# B&R Automation Studio project mappFramework (part 11)

#### Set_AuditMgr.c
```c
#include <bur/plctypes.h>
#include <fileio.h>

#ifdef _DEFAULT_INCLUDES
#include <AsDefault.h>
#endif

#include "UnitTest.h"
#include <stdbool.h>
#include <string.h>
#include <stdlib.h>

#define TIMEOUT_TEST_CASE									\
	if (cycleCount >= 1000)									\
	{														\
		char abortMessage[80];								\
		char substate[10];									\
		memset(abortMessage, 0, sizeof(abortMessage));		\
		memset(substate, 0, sizeof(substate));				\
		itoa(TestState, substate, 10);						\
		strcpy(abortMessage, "Timeout in State = ");		\
		strcat(abortMessage, substate);						\
		TEST_FAIL(abortMessage);							\
		TEST_DONE;											\
	}

_SETUP_SET(void)
{
	cycleCount = 0;

	TEST_DONE;
}

_TEARDOWN_SET(void)
{
	TEST_DONE;
}

_SETUP_TEST(void)
{
	ArrangeDelay = 0;
	ActDelay = 0;
	AssertDelay = 0;
	ArrangeSubState = 0;
	ActSubState = 0;
	AssertSubState = 0;
	SampleTemperature = 1;
	TestComparisonNumber = 0;
	TestState = TEST_ARRANGE;
	cycleCount = 0;

	TEST_DONE;
}

_TEARDOWN_TEST(void)
{
	ArrangeDelay = 0;
	ActDelay = 0;
	AssertDelay = 0;
	SampleTemperature = 1;
	TEST_DONE;
}

_CYCLIC_SET(void)
{
	cycleCount++;
}

_TEST ExportArchive(void)
{
	TIMEOUT_TEST_CASE;

	DirInfo_0.enable = 1;
	DirInfo_0.pDevice = (UDINT) "mappAuditFiles";
	DirInfo_0.pPath = 0;
	DirInfo(&DirInfo_0);

	switch (TestState)
	{
		case TEST_ARRANGE:
			// Force an audit to be generated
			switch (ArrangeSubState)
			{
				case 0:
					SampleTemperature++;
					TEST_BUSY_CONDITION(!HmiAudit.Status.ArchiveAvailable);
					ArrangeSubState = 1;
					break;

				case 1:
					ArrangeDelay += 1;												// This delay is compensating for the function block refreshing after finishing a command
					TEST_BUSY_CONDITION(ArrangeDelay <= DelayCycles);
					TestComparisonNumber = DirInfo_0.filenum;
					TestState = TEST_ACT;
					break;
			}
			break;

		case TEST_ACT:
			// Archive audit
			switch (ActSubState)
			{
				case 0:
					HmiAudit.Commands.ExportArchives = 1;
					TEST_ABORT_CONDITION(MpAuditTrailError);
					TEST_BUSY_CONDITION(!MpAuditTrailCmdDone);
					HmiAudit.Commands.ExportArchives = 0;
					ActSubState = 1;
					break;

				case 1:
					ActDelay += 1;													// This delay is compensating for the function block refreshing after finishing a command
					TEST_BUSY_CONDITION(ActDelay <= DelayCycles);
					TestState = TEST_ASSERT;
					break;
			}
			break;

		case TEST_ASSERT:
			TEST_ASSERT(TestComparisonNumber  < DirInfo_0.filenum);
			TEST_DONE;
			break;
	}

	TEST_BUSY;
}

_TEST AutomaticArchive(void)
{
	TIMEOUT_TEST_CASE;

	switch (TestState)
	{
		case TEST_ARRANGE:
			// Set automatic archive parameters prepare audit for generation
			switch (ArrangeSubState)
			{
				case 0:
					HmiAudit.Parameters.ArchiveSettings.Enable = 1;
					HmiAudit.Parameters.ArchiveSettings.FileType = mpAUDIT_FILE_TYPE_XML;
					HmiAudit.Parameters.ArchiveSettings.MaxSize = MAX_FILE_SIZE;
					HmiAudit.Parameters.ArchiveSettings.Mode = mpAUDIT_ARCHIVE_DAILY;
					HmiAudit.Parameters.ArchiveSettings.Hour = HOUR;
					HmiAudit.Parameters.ArchiveSettings.Minute = MINUTE;
					ArrangeSubState = 1;
					break;

				case 1:
					TestComparisonNumber = HmiAudit.Status.NumberOfArchives;
					ArrangeSubState = 2;
					break;

				case 2:
					ArrangeDelay += 1;
					TEST_BUSY_CONDITION(ArrangeDelay <= DelayCycles);
					TestState = TEST_ACT;
					break;
			}
			break;

		case TEST_ACT:
			// Archive audit
			switch (ActSubState)
			{
				case 0:
					SampleTemperature = SAMPLE_TEMP_VALUE;
					DTSetTime_0.DT1 = SET_TIME;
					DTSetTime_0.enable = 1;
					DTSetTime(&DTSetTime_0);
					ActSubState = 1;
					break;

				case 1:
					TON_0.PT = TIMER_LENGTH;
					TON_0.IN = 1;
					TON(&TON_0);
					if(TON_0.Q)
					{
						ActSubState = 2;
					}
					break;

				case 2:
					TestState = TEST_ASSERT;
					TON_0.IN = 0;
					TON(&TON_0);
					break;
			}
			break;

		case TEST_ASSERT:
			// Check save location for archive
			TEST_ASSERT(TestComparisonNumber + 1 <= HmiAudit.Status.NumberOfArchives);
			TEST_DONE;
			break;
	}
	TEST_BUSY;
}

/*
B+R UnitTest: This is generated code.
Do not edit! Do not move!
Description: UnitTest Testprogramm infrastructure (TestSet).
LastUpdated: 2023-02-06 16:23:26Z
By B+R UnitTest Helper Version: 2.0.1.59
*/
UNITTEST_FIXTURES(fixtures)
{
	new_TestFixture("ExportArchive", ExportArchive),
	new_TestFixture("AutomaticArchive", AutomaticArchive),
};

UNITTEST_CALLER_COMPLETE_EXPLICIT(Set_AuditMgr, "Set_AuditMgr", setupTest, teardownTest, fixtures, setupSet, teardownSet, cyclicSetCaller);
```

- Set_Common.c (reference to Logical/UnitTestVC4/Common/CommonUT/Set_Common.c)

### Package Logical/UnitTestVC4/AppAxis_1 - Package for mapp App_Axis1 Framework

### Program Logical/UnitTestVC4/AppAxis_1/AppAxisUnitTest (ANSIC) - Unit Tests for AppAxis_1

#### variables.var
```iecst
(********************************************************************
 * COPYRIGHT --
 ********************************************************************
 * Program: utTemplate_automated
 * File: variables.var
 * Author: -
 * Created: -
 ********************************************************************
 * Local variables of program utTemplate_automated
 ********************************************************************)
(*Describe the test*)
VAR
	Testsuite : UtMgrTestSuite := (Name:='AppAxis_1VC4',Description:='AppAxis_1 VC4 Unit Tests',MetaInformation:='Meta');
END_VAR
(*Variables used in the tests*)
VAR
	MpAlarmXListUIConnect : MpAlarmXListUIConnectType := (0); (*AlarmX list connection to the UI*)
	MpAlarmXListUI_0 : MpAlarmXListUI; (*MpAlarmXList instance*)
	MpAlarmXAcknowledgeAll_0 : MpAlarmXAcknowledgeAll;
	StartingActiveAlarms : UDINT;
	StartingPendingAlarms : UDINT;
	cycleCount : USINT;
	StartPosition : LREAL;
	maxVelocity : REAL;
END_VAR
```

#### autoGeneratedFile.c
```c
/*
B+R UnitTest: This is generated code.
Do not edit! Do not move!
Description: UnitTest Testprogramm infrastructure (List of TestSets).
LastUpdated: 2022-11-08 14:30:25Z
By B+R UnitTest Helper Version: 2.0.1.59
*/
#include "UnitTest.h"

UNITTEST_TESTSET_DECLARATION  Set_Common;
UNITTEST_TESTSET_DECLARATION  Set_ManualTests;
UNITTEST_TESTSET_DECLARATION  Set_AutomaticTests;

UNITTEST_TESTSET_FIXTURES(utTestSets)
{
	new_TestSet(Set_Common),
	new_TestSet(Set_ManualTests),
	new_TestSet(Set_AutomaticTests),
};
UNTITTEST_TESTSET_HANDLER();
```

#### Set_AutomaticTests.c
```c
#include <bur/plctypes.h>

#ifdef _DEFAULT_INCLUDES
#include <AsDefault.h>
#endif

#include "UnitTest.h"
#include <stdbool.h>
#include <string.h>
#include <math.h>
#include <stdlib.h>

#define MAX(x, y) (((x) > (y)) ? (x) : (y))

#define TIMEOUT_TEST_CASE									\
	if (cycleCount >= 254)									\
	{														\
		char abortMessage[80];								\
		char substate[10];									\
		memset(abortMessage, 0, sizeof(abortMessage));		\
		memset(substate, 0, sizeof(substate));				\
		itoa(ActSubState, substate, 10);					\
		strcpy(abortMessage, "Timeout in ActSubState = ");	\
		strcat(abortMessage, substate);						\
		TEST_FAIL(abortMessage);							\
		TEST_DONE;											\
	}

_SETUP_SET(void)
{
	TEST_DONE;
}

_TEARDOWN_SET(void)
{
	TEST_DONE;
}

_SETUP_TEST(void)
{
	cycleCount = 0;
	ArrangeSubState = 0;
	ActSubState = 0;
	AssertSubState = 0;
	TestState = TEST_ARRANGE;

	maxVelocity = 0.0;
	TEST_DONE;
}

_TEARDOWN_TEST(void)
{
	AxisControl.Command.JogNegative = false;
	AxisControl.Command.JogPositive = false;
	AxisControl.Command.Abort = false;
	AxisControl.Command.LoadRecipeParameters = false;
	AxisControl.Command.MoveAbsolute = false;
	AxisControl.Command.MoveAdditive = false;
	AxisControl.Command.MoveToStart = false;
	AxisControl.Command.MoveVelocity = false;
	AxisControl.Command.Reference = false;
	AxisControl.Command.Reset = false;
	AxisControl.Command.SaveRecipeParameters = false;
	AxisControl.Command.Start = false;
	AxisControl.Command.Stop = false;
	AxisControl.Command.UpdatePreviewParameters = false;
	AxisControl.Command.UpdateVelocity = false;

	if ((AxisControl.Status.ErrorActive == true) || (MpAlarmXCoreAxis.PendingAlarms > 0))
	{
		AxisControl.Command.Reset = true;
		MpAlarmXAcknowledgeAll_0.Execute = true;
	}
	TEST_BUSY_CONDITION(AxisControl.Status.ErrorActive);
	AxisControl.Command.Reset = false;
	if (abs(AxisControl.Status.Velocity) > 0.01)
		AxisControl.Command.Stop = true;
	TEST_BUSY_CONDITION(abs(AxisControl.Status.Velocity > 0.01));
	TEST_BUSY_CONDITION(AxisControl.Status.Busy);
	AxisControl.Command.Stop = false;

	TEST_DONE;
}

_CYCLIC_SET(void)
{
	cycleCount++;
	MpAlarmXAcknowledgeAll_0.MpLink = &gMpLinkAlarmXCoreAppAxis_1;
	MpAlarmXAcknowledgeAll_0.Enable = true;
	MpAlarmXAcknowledgeAll(&MpAlarmXAcknowledgeAll_0);
	MpAlarmXAcknowledgeAll_0.Execute = false;
}

_TEST Start(void)
{
	TIMEOUT_TEST_CASE
	switch (TestState)
	{
		case TEST_ARRANGE:
			AxisControl.Parameters.Velocity = 40;
			TestState = TEST_ACT;
			break;

		case TEST_ACT:
			maxVelocity = MAX(AxisControl.Status.Velocity, maxVelocity);
			switch (ActSubState)
			{
				case 0:
					AxisControl.Command.Start = true;
					TEST_BUSY_CONDITION(!AxisControl.Status.Busy);
					ActSubState = 1;
					break;

				case 1:
					TEST_BUSY_CONDITION(cycleCount < 30);
					TestState = TEST_ASSERT;
					break;
			}
			break;

		case TEST_ASSERT:
			TEST_ASSERT_FLOAT_WITHIN(0.1, 40.0, maxVelocity);
			TEST_DONE;
			break;
	}
	TEST_BUSY;
}

_TEST UpdateVelocity(void)
{
	TIMEOUT_TEST_CASE
	switch (TestState)
	{
		case TEST_ARRANGE:
			AxisControl.Parameters.Velocity = 40;
			TestState = TEST_ACT;
			break;

		case TEST_ACT:
			maxVelocity = MAX(AxisControl.Status.Velocity, maxVelocity);
			switch (ActSubState)
			{
				case 0:
					AxisControl.Command.Start = true;
					TEST_BUSY_CONDITION(!AxisControl.Status.Busy);
					ActSubState = 1;
					break;

				case 1:
					TEST_BUSY_CONDITION(cycleCount < 30);
					TEST_ASSERT_FLOAT_WITHIN(0.1, 40.0, maxVelocity);
					AxisControl.Command.UpdateVelocity = true;
					AxisControl.Parameters.Velocity = 60;
					ActSubState = 2;
					break;

				case 2:
					TEST_BUSY_CONDITION(cycleCount < 60);
					TestState = TEST_ASSERT;
					break;
			}
			break;

		case TEST_ASSERT:
			TEST_ASSERT_FLOAT_WITHIN(0.1, 60.0, maxVelocity);
			TEST_DONE;
			break;
	}
	TEST_BUSY;
}

_TEST ZeroVelocity(void)
{
	TIMEOUT_TEST_CASE
	switch (TestState)
	{
		case TEST_ARRANGE:
			AxisControl.Parameters.Velocity = 0;
			TestState = TEST_ACT;
			break;

		case TEST_ACT:
			maxVelocity = MAX(AxisControl.Status.Velocity, maxVelocity);
			switch (ActSubState)
			{
				case 0:
					AxisControl.Command.Start = true;
					TEST_BUSY_CONDITION(!AxisControl.Status.Busy);
					ActSubState = 1;
					break;

				case 1:
					TEST_BUSY_CONDITION(cycleCount < 10);
					TestState = TEST_ASSERT;
					break;
			}
			break;

		case TEST_ASSERT:
			TEST_ASSERT(AxisControl.Status.ErrorActive);
			TEST_ASSERT_EQUAL_INT(1, MpAlarmXCoreAxis.PendingAlarms);
			TEST_ASSERT_FLOAT_WITHIN(0.1, 0.0, maxVelocity);
			TEST_DONE;
			break;
	}
	TEST_BUSY;
}

/*
B+R UnitTest: This is generated code.
Do not edit! Do not move!
Description: UnitTest Testprogramm infrastructure (TestSet).
LastUpdated: 2022-11-08 14:33:54Z
By B+R UnitTest Helper Version: 2.0.1.59
*/
UNITTEST_FIXTURES(fixtures)
{
	new_TestFixture("Start", Start),
	new_TestFixture("UpdateVelocity", UpdateVelocity),
	new_TestFixture("ZeroVelocity", ZeroVelocity),
};

UNITTEST_CALLER_COMPLETE_EXPLICIT(Set_AutomaticTests, "Set_AutomaticTests", setupTest, teardownTest, fixtures, setupSet, teardownSet, cyclicSetCaller);
```

#### Set_ManualTests.c
```c
#include <bur/plctypes.h>

#ifdef _DEFAULT_INCLUDES
#include <AsDefault.h>
#endif

#include "UnitTest.h"
#include <stdbool.h>
#include <string.h>
#include <math.h>
#include <stdlib.h>

#define MAX(x, y) (((x) > (y)) ? (x) : (y))

#define TIMEOUT_TEST_CASE									\
	if (cycleCount >= 254)									\
	{														\
		char abortMessage[80];								\
		char substate[10];									\
		memset(abortMessage, 0, sizeof(abortMessage));		\
		memset(substate, 0, sizeof(substate));				\
		itoa(ActSubState, substate, 10);					\
		strcpy(abortMessage, "Timeout in ActSubState = ");	\
		strcat(abortMessage, substate);						\
		TEST_FAIL(abortMessage);							\
		TEST_DONE;											\
	}

_SETUP_SET(void)
{
	TEST_DONE;
}

_TEARDOWN_SET(void)
{
	TEST_DONE;
}

_SETUP_TEST(void)
{
	cycleCount = 0;
	ArrangeSubState = 0;
	ActSubState = 0;
	AssertSubState = 0;
	TestState = TEST_ARRANGE;

	maxVelocity = 0.0;

	TEST_DONE;
}

_TEARDOWN_TEST(void)
{
	AxisControl.Command.JogNegative = false;
	AxisControl.Command.JogPositive = false;
	AxisControl.Command.Abort = false;
	AxisControl.Command.LoadRecipeParameters = false;
	AxisControl.Command.MoveAbsolute = false;
	AxisControl.Command.MoveAdditive = false;
	AxisControl.Command.MoveToStart = false;
	AxisControl.Command.MoveVelocity = false;
	AxisControl.Command.Reference = false;
	AxisControl.Command.Reset = false;
	AxisControl.Command.SaveRecipeParameters = false;
	AxisControl.Command.Start = false;
	AxisControl.Command.Stop = false;
	AxisControl.Command.UpdatePreviewParameters = false;
	AxisControl.Command.UpdateVelocity = false;

	if ((AxisControl.Status.ErrorActive == true) || (MpAlarmXCoreAxis.PendingAlarms > 0))
	{
		AxisControl.Command.Reset = true;
		MpAlarmXAcknowledgeAll_0.Execute = true;
	}
	TEST_BUSY_CONDITION(AxisControl.Status.ErrorActive);
	AxisControl.Command.Reset = false;
	if (abs(AxisControl.Status.Velocity) > 0.01)
		AxisControl.Command.Stop = true;
	TEST_BUSY_CONDITION(abs(AxisControl.Status.Velocity > 0.01));
	TEST_BUSY_CONDITION(AxisControl.Status.Busy);
	AxisControl.Command.Stop = false;

	TEST_DONE;
}

_CYCLIC_SET(void)
{
	cycleCount++;

	MpAlarmXListUI_0.Enable = true;
	MpAlarmXListUI_0.UIConnect = &MpAlarmXListUIConnect;
	MpAlarmXListUI_0.MpLink = &gMpLinkAlarmXCoreAppAxis_1;
	MpAlarmXListUI_0.UISetup.AlarmListScrollWindow = 10;
	MpAlarmXListUI_0.UISetup.AlarmListSize = 50;
	strcpy(MpAlarmXListUI_0.UISetup.TimeStampPattern, "%Y %m %d %H:%M:%S");
	MpAlarmXListUI(&MpAlarmXListUI_0);

	MpAlarmXAcknowledgeAll_0.MpLink = &gMpLinkAlarmXCoreAppAxis_1;
	MpAlarmXAcknowledgeAll_0.Enable = true;
	MpAlarmXAcknowledgeAll(&MpAlarmXAcknowledgeAll_0);
	TEST_BUSY_CONDITION(MpAlarmXAcknowledgeAll_0.CommandBusy);
	MpAlarmXAcknowledgeAll_0.Execute = false;

}

_TEST PowerOn(void)
{
	TIMEOUT_TEST_CASE
	switch (TestState)
	{
		case TEST_ARRANGE:
			TestState = TEST_ACT;
			break;

		case TEST_ACT:
			switch (ActSubState)
			{
				case 0:
					AxisControl.Command.Power = true;
					ActSubState = 1;
					break;
				case 1:
					TEST_BUSY_CONDITION(AxisControl.Status.Busy == true);
					TestState = TEST_ASSERT;
					break;
			}
			break;

		case TEST_ASSERT:
			TEST_ASSERT(AxisControl.Status.IsPowered);
			TEST_DONE;
			break;
	}
	TEST_BUSY;
}

_TEST Homing(void)
{
	TIMEOUT_TEST_CASE
	switch (TestState)
	{
		case TEST_ARRANGE:
			TestState = TEST_ACT;
			break;

		case TEST_ACT:
			switch (ActSubState)
			{
				case 0:
					AxisControl.Command.Reference = true;
					ActSubState = 1;
					break;
				case 1:
					TEST_BUSY_CONDITION(AxisControl.Status.IsHomed == false);
					TEST_BUSY_CONDITION(!AxisControl.Status.Busy);
					ActSubState = 2;
					break;

				case 2:
					TEST_BUSY_CONDITION(AxisControl.Status.Busy);
					TestState = TEST_ASSERT;
					break;
			}
			break;

		case TEST_ASSERT:
			TEST_ASSERT(AxisControl.Status.IsHomed);
			TEST_ASSERT_DOUBLE_WITHIN(0.0001, 0.0, AxisControl.Status.Position);
			TEST_DONE;
			break;
	}
	TEST_BUSY;
}

_TEST JogPositive(void)
{
	TIMEOUT_TEST_CASE
	switch (TestState)
	{
		case TEST_ARRANGE:
			TestState = TEST_ACT;
			break;

		case TEST_ACT:
			switch (ActSubState)
			{
				case 0:
					AxisControl.Command.JogPositive = true;
					AxisControl.Parameters.JogVelocity = 50;
					ActSubState = 1;
					break;
				case 1:
					TEST_BUSY_CONDITION(AxisControl.Status.Velocity <= 49.0);
					TestState = TEST_ASSERT;
					break;
			}
			break;

		case TEST_ASSERT:
			TEST_ASSERT_FLOAT_WITHIN(0.1, 50.0, AxisControl.Status.Velocity);
			TEST_DONE;
			break;
	}
	TEST_BUSY;
}

_TEST JogNegative(void)
{
	TIMEOUT_TEST_CASE
	switch (TestState)
	{
		case TEST_ARRANGE:
			TestState = TEST_ACT;
			break;

		case TEST_ACT:
			switch (ActSubState)
			{
				case 0:
					AxisControl.Command.JogNegative = true;
					AxisControl.Parameters.JogVelocity = 50;
					ActSubState = 1;
					break;
				case 1:
					TEST_BUSY_CONDITION(AxisControl.Status.Velocity >= -49.0);
					TestState = TEST_ASSERT;
					break;
			}
			break;

		case TEST_ASSERT:
			TEST_ASSERT_FLOAT_WITHIN(0.1, -50.0, AxisControl.Status.Velocity);
			TEST_DONE;
			break;
	}
	TEST_BUSY;
}

_TEST MoveAbsolute(void)
{
	TIMEOUT_TEST_CASE
	switch (TestState)
	{
		case TEST_ARRANGE:
			AxisControl.Parameters.Position = 10;
			AxisControl.Parameters.Velocity = 40;
			TestState = TEST_ACT;
			break;

		case TEST_ACT:
			maxVelocity = MAX(AxisControl.Status.Velocity, maxVelocity);
			switch (ActSubState)
			{
				case 0:
					AxisControl.Command.MoveAbsolute = true;
					TEST_BUSY_CONDITION(!AxisControl.Status.Busy);
					ActSubState = 1;
					break;
				case 1:
					TEST_BUSY_CONDITION(AxisControl.Status.Busy);
					AxisControl.Command.MoveAbsolute = false;
					TestState = TEST_ASSERT;
					break;
			}
			break;

		case TEST_ASSERT:
			TEST_ASSERT_FLOAT_WITHIN(0.1, 40.0, maxVelocity);
			TEST_ASSERT_FLOAT_WITHIN(0.01, 10.0, AxisControl.Status.Position);
			TEST_DONE;
			break;
	}
	TEST_BUSY;
}

_TEST MoveAdditive(void)
{
	TIMEOUT_TEST_CASE
	switch (TestState)
	{
		case TEST_ARRANGE:
			AxisControl.Parameters.Distance = 5;
			AxisControl.Parameters.Velocity = 30;
			StartPosition = AxisControl.Status.Position;
			TestState = TEST_ACT;
			break;

		case TEST_ACT:
			maxVelocity = MAX(AxisControl.Status.Velocity, maxVelocity);
			switch (ActSubState)
			{
				case 0:
					AxisControl.Command.MoveAdditive = true;
					TEST_BUSY_CONDITION(!AxisControl.Status.Busy);
					ActSubState = 1;
					break;
				case 1:
					TEST_BUSY_CONDITION(AxisControl.Status.Busy);
					AxisControl.Command.MoveAbsolute = false;
					TestState = TEST_ASSERT;
					break;
			}
			break;

		case TEST_ASSERT:
			TEST_ASSERT_FLOAT_WITHIN(0.1, 30.0, maxVelocity);
			TEST_ASSERT_FLOAT_WITHIN(0.01, StartPosition + 5.0, AxisControl.Status.Position);
			TEST_DONE;
			break;
	}
	TEST_BUSY;
}

_TEST MoveVelocity(void)
{
	TIMEOUT_TEST_CASE
	switch (TestState)
	{
		case TEST_ARRANGE:
			AxisControl.Parameters.Velocity = 25;
			TestState = TEST_ACT;
			break;

		case TEST_ACT:
			maxVelocity = MAX(AxisControl.Status.Velocity, maxVelocity);
			switch (ActSubState)
			{
				case 0:
					AxisControl.Command.MoveVelocity = true;
					TEST_BUSY_CONDITION(!AxisControl.Status.Busy);
					ActSubState = 1;
					break;
				case 1:
					TEST_BUSY_CONDITION(cycleCount < 30);
					TestState = TEST_ASSERT;
					break;
			}
			break;

		case TEST_ASSERT:
			TEST_ASSERT_FLOAT_WITHIN(0.1, 25.0, maxVelocity);
			TEST_DONE;
			break;
	}
	TEST_BUSY;
}

_TEST MoveJogPositiveStop(void)
{
	TIMEOUT_TEST_CASE
	switch (TestState)
	{
		case TEST_ARRANGE:
			AxisControl.Parameters.JogVelocity = 25;
			TestState = TEST_ACT;
			break;

		case TEST_ACT:
			maxVelocity = MAX(AxisControl.Status.Velocity, maxVelocity);
			switch (ActSubState)
			{
				case 0:
					AxisControl.Command.JogPositive = true;
					TEST_BUSY_CONDITION(!AxisControl.Status.Busy);
					ActSubState = 1;
					break;
				case 1:
					TEST_BUSY_CONDITION(cycleCount < 30);
					AxisControl.Command.JogPositive = false;
					ActSubState = 2;
					break;
				case 2:
					TEST_BUSY_CONDITION(AxisControl.Status.Busy);
					TestState = TEST_ASSERT;
					break;
			}
			break;

		case TEST_ASSERT:
			TEST_ASSERT_FLOAT_WITHIN(0.1, 0.0, AxisControl.Status.Velocity);
			TEST_DONE;
			break;
	}
	TEST_BUSY;
}

_TEST MoveJogNegativeStop(void)
{
	TIMEOUT_TEST_CASE
	switch (TestState)
	{
		case TEST_ARRANGE:
			AxisControl.Parameters.JogVelocity = 25;
			TestState = TEST_ACT;
			break;

		case TEST_ACT:
			maxVelocity = MAX(AxisControl.Status.Velocity, maxVelocity);
			switch (ActSubState)
			{
				case 0:
					AxisControl.Command.JogNegative = true;
					TEST_BUSY_CONDITION(!AxisControl.Status.Busy);
					ActSubState = 1;
					break;
				case 1:
					TEST_BUSY_CONDITION(cycleCount < 30);
					AxisControl.Command.JogNegative = false;
					ActSubState = 2;
					break;
				case 2:
					TEST_BUSY_CONDITION(AxisControl.Status.Busy);
					TestState = TEST_ASSERT;
					break;
			}
			break;

		case TEST_ASSERT:
			TEST_ASSERT_FLOAT_WITHIN(0.1, 0.0, AxisControl.Status.Velocity);
			TEST_DONE;
			break;
	}
	TEST_BUSY;
}

_TEST MoveAbsoluteStop(void)
{
	TIMEOUT_TEST_CASE
	switch (TestState)
	{
		case TEST_ARRANGE:
			AxisControl.Parameters.Position = 1;
			AxisControl.Parameters.Velocity = 25;
			TestState = TEST_ACT;
			break;

		case TEST_ACT:
			maxVelocity = MAX(AxisControl.Status.Velocity, maxVelocity);
			switch (ActSubState)
			{
				case 0:
					AxisControl.Command.MoveAbsolute = true;
					TEST_BUSY_CONDITION(!AxisControl.Status.Busy);
					ActSubState = 1;
					break;
				case 1:
					TEST_BUSY_CONDITION(cycleCount < 30);
					AxisControl.Command.MoveAbsolute = false;
					AxisControl.Command.Stop = true;
					ActSubState = 2;
					break;
				case 2:
					TEST_BUSY_CONDITION(AxisControl.Status.Busy);
					TestState = TEST_ASSERT;
					break;
			}
			break;

		case TEST_ASSERT:
			TEST_ASSERT_FLOAT_WITHIN(0.1, 0.0, AxisControl.Status.Velocity);
			// check that we are not at the target position
			TEST_ASSERT(fabs(1.0 - AxisControl.Status.Position) > 0.01);
			TEST_DONE;
			break;
	}
	TEST_BUSY;
}

_TEST MoveAdditiveStop(void)
{
	TIMEOUT_TEST_CASE
	switch (TestState)
	{
		case TEST_ARRANGE:
			AxisControl.Parameters.Distance = 10;
			AxisControl.Parameters.Velocity = 25;
			StartPosition = AxisControl.Status.Position;
			TestState = TEST_ACT;
			break;

		case TEST_ACT:
			maxVelocity = MAX(AxisControl.Status.Velocity, maxVelocity);
			switch (ActSubState)
			{
				case 0:
					AxisControl.Command.MoveAdditive = true;
					TEST_BUSY_CONDITION(!AxisControl.Status.Busy);
					ActSubState = 1;
					break;
				case 1:
					TEST_BUSY_CONDITION(cycleCount < 30);
					AxisControl.Command.MoveAdditive = false;
					AxisControl.Command.Stop = true;
					ActSubState = 2;
					break;
				case 2:
					TEST_BUSY_CONDITION(AxisControl.Status.Busy);
					TestState = TEST_ASSERT;
					break;
			}
			break;

		case TEST_ASSERT:
			TEST_ASSERT_FLOAT_WITHIN(0.1, 0.0, AxisControl.Status.Velocity);
			// check that we are not at the target position
			TEST_ASSERT(fabs((StartPosition + 10.0) - AxisControl.Status.Position) > 0.01);
			TEST_DONE;
			break;
	}
	TEST_BUSY;
}

_TEST MoveVelocityStop(void)
{
	TIMEOUT_TEST_CASE
	switch (TestState)
	{
		case TEST_ARRANGE:
			AxisControl.Parameters.Velocity = 25;
			TestState = TEST_ACT;
			break;

		case TEST_ACT:
			maxVelocity = MAX(AxisControl.Status.Velocity, maxVelocity);
			switch (ActSubState)
			{
				case 0:
					AxisControl.Command.MoveVelocity = true;
					TEST_BUSY_CONDITION(!AxisControl.Status.Busy);
					ActSubState = 1;
					break;
				case 1:
					TEST_BUSY_CONDITION(cycleCount < 30);
					AxisControl.Command.MoveVelocity = false;
					AxisControl.Command.Stop = true;
					ActSubState = 2;
					break;
				case 2:
					TEST_BUSY_CONDITION(AxisControl.Status.Busy);
					TestState = TEST_ASSERT;
					break;
			}
			break;

		case TEST_ASSERT:
			TEST_ASSERT_FLOAT_WITHIN(0.1, 0.0, AxisControl.Status.Velocity);
			TEST_DONE;
			break;
	}
	TEST_BUSY;
}

_TEST TriggerAlarm(void)
{
	TIMEOUT_TEST_CASE
	switch (TestState)
	{
		case TEST_ARRANGE:
			AxisControl.Parameters.Velocity = 10001;
			TestState = TEST_ACT;
			break;

		case TEST_ACT:
			maxVelocity = MAX(AxisControl.Status.Velocity, maxVelocity);
			switch (ActSubState)
			{
				case 0:
					AxisControl.Command.MoveVelocity = true;
					TEST_BUSY_CONDITION(!AxisControl.Status.Busy);
					ActSubState = 1;
					break;
				case 1:
					TEST_BUSY_CONDITION(cycleCount < 20);
					TestState = TEST_ASSERT;
					break;
			}
			break;

		case TEST_ASSERT:
			TEST_ASSERT_FLOAT_WITHIN(0.1, 0.0, AxisControl.Status.Velocity);
			TEST_ASSERT_FLOAT_WITHIN(0.1, 0.0, maxVelocity);
			TEST_ASSERT(AxisControl.Status.ErrorActive);
			TEST_ASSERT_EQUAL_INT(1, MpAlarmXCoreAxis.PendingAlarms);
			TEST_DONE;
			break;
	}
	TEST_BUSY;
}

_TEST ResetAlarm(void)
{
	TIMEOUT_TEST_CASE
	switch (TestState)
	{
		case TEST_ARRANGE:
			AxisControl.Parameters.Velocity = 10001;
			StartingPendingAlarms = MpAlarmXCoreAxis.PendingAlarms;
			TestState = TEST_ACT;
			break;

		case TEST_ACT:
			maxVelocity = MAX(AxisControl.Status.Velocity, maxVelocity);
			switch (ActSubState)
			{
				case 0:
					AxisControl.Command.MoveVelocity = true;
					TEST_BUSY_CONDITION(!AxisControl.Status.Busy);
					ActSubState = 1;
					break;
				case 1:
					TEST_BUSY_CONDITION(!AxisControl.Status.ErrorActive);
					TEST_BUSY_CONDITION(MpAlarmXCoreAxis.PendingAlarms == StartingPendingAlarms);
					AxisControl.Command.MoveVelocity = false;
					ActSubState = 2;
					break;
				case 2:
					// wait until the command is received by the axis task
					TEST_BUSY_CONDITION(State != STATE_RESETTING);
					AxisControl.Command.Reset = true;
					MpAlarmXAcknowledgeAll_0.Execute = true;
					ActSubState = 3;
					break;
				case 3:
					TEST_BUSY_CONDITION(AxisControl.Status.Busy);
					TestState = TEST_ASSERT;
					break;
			}
			break;

		case TEST_ASSERT:
			TEST_ASSERT(!AxisControl.Status.ErrorActive);
			TEST_ASSERT_EQUAL_INT(0, MpAlarmXCoreAxis.PendingAlarms);
			TEST_DONE;
			break;
	}
	TEST_BUSY;
}

_TEST UpdateVelocity(void)
{
	TIMEOUT_TEST_CASE
	switch (TestState)
	{
		case TEST_ARRANGE:
			AxisControl.Parameters.Velocity = 40;
			TestState = TEST_ACT;
			break;

		case TEST_ACT:
			maxVelocity = MAX(AxisControl.Status.Velocity, maxVelocity);
			switch (ActSubState)
			{
				case 0:
					AxisControl.Command.MoveVelocity = true;
					TEST_BUSY_CONDITION(!AxisControl.Status.Busy);
					ActSubState = 1;
					break;
				case 1:
					TEST_BUSY_CONDITION(cycleCount < 30);
					TEST_ASSERT_FLOAT_WITHIN(0.1, 40.0, maxVelocity);
					AxisControl.Command.UpdateVelocity = true;
					AxisControl.Parameters.Velocity = 60;
					ActSubState = 2;
					break;
				case 2:
					TEST_BUSY_CONDITION(cycleCount < 60);
					TestState = TEST_ASSERT;
					break;
			}
			break;

		case TEST_ASSERT:
			// update velocity should not affect manual moves
			TEST_ASSERT_FLOAT_WITHIN(0.1, 40.0, maxVelocity);
			TEST_DONE;
			break;
	}
	TEST_BUSY;
}

/*
B+R UnitTest: This is generated code.
Do not edit! Do not move!
Description: UnitTest Testprogramm infrastructure (TestSet).
LastUpdated: 2022-11-15 16:02:39Z
By B+R UnitTest Helper Version: 2.0.1.59
*/
UNITTEST_FIXTURES(fixtures)
{
	new_TestFixture("PowerOn", PowerOn),
	new_TestFixture("Homing", Homing),
	new_TestFixture("JogPositive", JogPositive),
	new_TestFixture("JogNegative", JogNegative),
	new_TestFixture("MoveAbsolute", MoveAbsolute),
	new_TestFixture("MoveAdditive", MoveAdditive),
	new_TestFixture("MoveVelocity", MoveVelocity),
	new_TestFixture("MoveJogPositiveStop", MoveJogPositiveStop),
	new_TestFixture("MoveJogNegativeStop", MoveJogNegativeStop),
	new_TestFixture("MoveAbsoluteStop", MoveAbsoluteStop),
	new_TestFixture("MoveAdditiveStop", MoveAdditiveStop),
	new_TestFixture("MoveVelocityStop", MoveVelocityStop),
	new_TestFixture("TriggerAlarm", TriggerAlarm),
	new_TestFixture("ResetAlarm", ResetAlarm),
	new_TestFixture("UpdateVelocity", UpdateVelocity),
};

UNITTEST_CALLER_COMPLETE_EXPLICIT(Set_ManualTests, "Set_ManualTests", setupTest, teardownTest, fixtures, setupSet, teardownSet, cyclicSetCaller);
```

#### testSuite.c
```c
/********************************************************************
 * COPYRIGHT --
 ********************************************************************
 * Program: -
 * Author:
 * Created:
 ********************************************************************
 * Test registration and handshake
 ********************************************************************/

#include <bur/plctypes.h>

#ifdef _DEFAULT_INCLUDES
#include <AsDefault.h>
#endif

#include "UnitTest.h"
#include <string.h>
#include <stdbool.h>

void _INIT initTestSuite(void)
{
	Testsuite.Enable = 1;
	utInit(&Testsuite);

	CommonTestsuite.Enable = 1;
	utInit(&CommonTestsuite);

	strcpy((char*)&FileDeviceName, "");
	strcpy((char*)&TextNameSpace, "Axis/Alarms");
	strcpy((char*)&TextID, "ReferenceRequired");
}

void _CYCLIC cyclicWithTest(void)
{
	utCyclic(&Testsuite);

	if (Testsuite.Informational.LastKnownPassedLocation.TestCaseName != 0)
		strcpy((char*)&LastTestCase, (char*)Testsuite.Informational.LastKnownPassedLocation.TestCaseName);
	if (Testsuite.Informational.LastKnownPassedLocation.TestSetName != 0)
		strcpy((char*)&LastTestSet, (char*)Testsuite.Informational.LastKnownPassedLocation.TestSetName);
	if (Testsuite.Informational.LastKnownPassedLocation.File != 0)
		strcpy((char*)&LastTestFile, (char*)Testsuite.Informational.LastKnownPassedLocation.File);
}

void _EXIT exitTestSuite(void)
{
	utExit(&Testsuite);
}
```

### Package Logical/UnitTestVC4/Backup - Package for mapp Backup Framework

### Program Logical/UnitTestVC4/Backup/BackupUnitTest (ANSIC)

- BackupMgr.typ (reference to Logical/Infrastructure/VC4/Backup/BackupMgr/BackupMgr.typ)

- BackupMgr.var (reference to Logical/Infrastructure/VC4/Backup/BackupMgr/BackupMgr.var)

#### variables.var - Name the suite and add PVs for the program
```iecst
(********************************************************************
 * COPYRIGHT --
 ********************************************************************
 * Program: utTemplate_automated
 * File: variables.var
 * Author: -
 * Created: -
 ********************************************************************
 * Local variables of program utTemplate_automated
 ********************************************************************)
(*Describe the test*)
VAR
	Testsuite : UtMgrTestSuite := (Name:='BackupMgrVC4',Description:='BackupMgr VC4 Unit Tests',MetaInformation:='Meta');
END_VAR
(*Variables used in the tests*)
```

#### testSuite.c
```c
/********************************************************************
 * COPYRIGHT --
 ********************************************************************
 * Program: -
 * Author:
 * Created:
 ********************************************************************
 * Test registration and handshake
 ********************************************************************/

#include <bur/plctypes.h>

#ifdef _DEFAULT_INCLUDES
#include <AsDefault.h>
#endif

#include "UnitTest.h"
#include <string.h>

void _INIT initTestSuite(void)
{
	Testsuite.Enable = 1;
	utInit(&Testsuite);

	CommonTestsuite.Enable = 1;
	utInit(&CommonTestsuite);

	strcpy((char*)&FileDeviceName, "mappBackupFiles");
	strcpy((char*)&TextNameSpace, "mappFramework/Backup/Alarms");
	strcpy((char*)&TextID, "CreateFailed");

}

void _CYCLIC cyclicWithTest(void)
{
	utCyclic(&Testsuite);
}

void _EXIT exitTestSuite(void)
{
	utExit(&Testsuite);
}
```

#### Set_BackupMgr.c
```c
#include <bur/plctypes.h>

#ifdef _DEFAULT_INCLUDES
#include <AsDefault.h>
#endif

#include "UnitTest.h"
#include <stdbool.h>
#include <string.h>

_SETUP_SET(void)
{
	TEST_DONE;
}

_TEARDOWN_SET(void)
{
	TEST_DONE;
}

_SETUP_TEST(void)
{
	TEST_DONE;
}

_TEARDOWN_TEST(void)
{
	TEST_DONE;
}

/*
B+R UnitTest: This is generated code.
Do not edit! Do not move!
Description: UnitTest Testprogramm infrastructure (TestSet).
LastUpdated: 2022-09-22 14:29:52Z
By B+R UnitTest Helper Version: 2.0.1.59
*/
UNITTEST_FIXTURES(fixtures)
{
};

UNITTEST_CALLER_COMPLETE_EXPLICIT(Set_BackupMgr, "Set_BackupMgr", setupTest, teardownTest, fixtures, setupSet, teardownSet, 0);
```

- Set_Common.c (reference to Logical/UnitTestVC4/Common/CommonUT/Set_Common.c)

### Package Logical/UnitTestVC4/File - Package for mapp File Framework

### Program Logical/UnitTestVC4/File/FileUnitTest (ANSIC) - Unit Tests for FileMgr

- FileMgr.typ (reference to Logical/Infrastructure/VC4/File/FileMgr/FileMgr.typ)

- FileMgr.var (reference to Logical/Infrastructure/VC4/File/FileMgr/FileMgr.var)

- Set_Common.c (reference to Logical/UnitTestVC4/Common/CommonUT/Set_Common.c)

#### variables.var - Name the suite and add PVs for the program
```iecst
(********************************************************************
 * COPYRIGHT --
 ********************************************************************
 * Program: utTemplate_automated
 * File: variables.var
 * Author: -
 * Created: -
 ********************************************************************
 * Local variables of program utTemplate_automated
 ********************************************************************)
(*Describe the test*)
VAR
	Testsuite : UtMgrTestSuite := (Name:='FileMgrVC4',Description:='FileMgr VC4 Unit Tests',Type:=utMgrTEST_TYPE_C,MetaInformation:='Meta');
END_VAR
(*Variables used in the tests*)
VAR
	cycleCount : {REDUND_UNREPLICABLE} UINT;
	HmiFile_UT : FileHmiInterfaceType; (*HMI interface structure*)
	FileName : STRING[24];
	FileNumber : USINT;
	SetupState : USINT;
	FileCreate_UT : FileCreate;
	FileClose_UT : FileClose;
	NumberOfFiles : UINT;
	CurrentFile : UINT;
	DirInfo_UT : DirInfo;
	fileInfo : fiDIR_READ_DATA;
	DirRead_UT : DirRead;
	FileWrite_UT : FileWrite;
	testData : {REDUND_UNREPLICABLE} STRING[1023] := 'testing data';
	FileDelete_UT : FileDelete;
	NameMatch : BOOL;
	DirName : STRING[255] := 'FileTestDir';
	CreateFileName : STRING[255] := 'FileTestFile.xml';
	FileCreate_0 : FileCreate;
	FileClose_0 : FileClose;
	CopiedFileName : STRING[255] := 'FileTestFile(1).xml';
	CopiedDirName : STRING[255] := 'FileTestDir(1)';
	NewFileName : STRING[255] := 'FileRename.xml';
	NewDirName : STRING[255] := 'DirRename';
	InNewLocation : BOOL;
	InOldLocation : BOOL;
	CopiedNewFileName : STRING[255] := 'FileRename(1).xml';
	CopiedNewDirName : STRING[255] := 'DirRename(1)';
	MultiSelectFileCopy : BOOL;
	MultiSelectDirCopy : BOOL;
END_VAR
```

#### testSuite.c
```c
/********************************************************************
 * COPYRIGHT --
 ********************************************************************
 * Program: -
 * Author:
 * Created:
 ********************************************************************
 * Test registration and handshake
 ********************************************************************/

#include <bur/plctypes.h>

#ifdef _DEFAULT_INCLUDES
#include <AsDefault.h>
#endif
#include <string.h>

#include "UnitTest.h"

void _INIT initTestSuite(void)
{
	Testsuite.Enable = 1;
	utInit(&Testsuite);

	CommonTestsuite.Enable = 1;
	utInit(&CommonTestsuite);

	strcpy((char*)&TextNameSpace, "mappFramework/File/Alarms");
	strcpy((char*)&TextID, "DeviceNotFound");
	strcpy(FileDeviceName, "mappUserXFiles");
}

void _CYCLIC cyclicWithTest(void)
{
	utCyclic(&Testsuite);
	if (Testsuite.Informational.LastKnownPassedLocation.TestCaseName != 0)
		strcpy((char*)&LastTestCase, (char*)Testsuite.Informational.LastKnownPassedLocation.TestCaseName);
	if (Testsuite.Informational.LastKnownPassedLocation.TestSetName != 0)
		strcpy((char*)&LastTestSet, (char*)Testsuite.Informational.LastKnownPassedLocation.TestSetName);
	if (Testsuite.Informational.LastKnownPassedLocation.File != 0)
		strcpy((char*)&LastTestFile, (char*)Testsuite.Informational.LastKnownPassedLocation.File);
}

void _EXIT exitTestSuite(void)
{
	utExit(&Testsuite);
}
```

#### Set_FileMgr.c
```c
#include <bur/plctypes.h>

#ifdef _DEFAULT_INCLUDES
#include <AsDefault.h>
#endif

#include "UnitTest.h"
#include <stdbool.h>
#include <string.h>
#include <stdlib.h>

#define TIMEOUT_TEST_CASE								\
	if (cycleCount >= 1000)								\
	{													\
	char abortMessage[80];								\
	char substate[10];									\
	memset(abortMessage, 0, sizeof(abortMessage));		\
	memset(substate, 0, sizeof(substate));				\
	itoa(TestState, substate, 10);						\
	strcpy(abortMessage, "Timeout in State = ");		\
	strcat(abortMessage, substate);						\
	TEST_FAIL(abortMessage);							\
	TEST_DONE;											\
	}

_SETUP_SET(void)
{
	TestState = 0;
	FileNumber = 0;

	HmiFile_UT.Parameters.Fifo.Enable = false;
	HmiFile_UT.Parameters.Fifo.ScanInterval = 60;
	strcpy(HmiFile_UT.Parameters.Fifo.DeviceName, "mappUserXFiles");

	switch (SetupState)
	{
		case 0:
			TEST_BUSY_CONDITION(HmiFile_UT.Status.DeleteStep != FILE_DISABLED);
			for (USINT i=0; i<sizeof(HmiFile_UT.Status.FifoSelect)/sizeof(HmiFile_UT.Status.FifoSelect[0]); i++)
			{
				TEST_BUSY_CONDITION(HmiFile_UT.Status.FifoSelect[i] != 0);
			}

			DirInfo_UT.enable = true;
			DirInfo_UT.pDevice = (UDINT)&"mappUserXFiles";
			DirInfo_UT.pPath = (UDINT)&"";
			DirInfo(&DirInfo_UT);
			TEST_BUSY_CONDITION(DirInfo_UT.status == 65535);
			TEST_ABORT_CONDITION(DirInfo_UT.status != 0);
			NumberOfFiles = DirInfo_UT.filenum;
			CurrentFile = 0;
			SetupState = (NumberOfFiles == 0) ? 100 : 1;
			break;

		case 1:
			DirRead_UT.enable = true;
			DirRead_UT.pDevice = DirInfo_UT.pDevice;
			DirRead_UT.entry = 0;
			DirRead_UT.option = fiFILE;
			DirRead_UT.pData = (UDINT)&fileInfo;
			DirRead_UT.data_len = sizeof(fileInfo);
			DirRead(&DirRead_UT);
			TEST_BUSY_CONDITION(DirRead_UT.status == 65535);
			TEST_ABORT_CONDITION(DirRead_UT.status != 0);
			SetupState = 2;
			break;

		case 2:
			FileDelete_UT.enable = true;
			FileDelete_UT.pDevice = DirInfo_UT.pDevice;
			FileDelete_UT.pName = (UDINT)&fileInfo.Filename;
			FileDelete(&FileDelete_UT);
			TEST_BUSY_CONDITION(FileDelete_UT.status == 65535);
			TEST_ABORT_CONDITION(FileDelete_UT.status != 0);

			CurrentFile++;
			SetupState = (CurrentFile >= NumberOfFiles) ? 100 : 1;
			break;

		case 10:
			TEST_BUSY_CONDITION(MpFileManagerUIConnect_FIFO.Status == mpFILE_UI_STATUS_IDLE);
			MpFileManagerUIConnect_FIFO.File.Refresh = true;
			TEST_BUSY_CONDITION(MpFileManagerUIConnect_FIFO.Status == mpFILE_UI_STATUS_IDLE);
			MpFileManagerUIConnect_FIFO.File.Refresh = false;
			SetupState = 11;
			break;

		case 11:
			TEST_BUSY_CONDITION(MpFileManagerUIConnect_FIFO.Status != mpFILE_UI_STATUS_IDLE);
			SetupState = 100;
			break;

		case 100:
			TEST_DONE;
	}
	TEST_BUSY;
}

_TEARDOWN_SET(void)
{
	/* TODO:  add code running after test set here */
	TEST_DONE;
}

bool FileIdleOrDisabled(void) {
	return ((HmiFile_UT.Status.DeleteStep == FILE_DELETE_WAIT) || (HmiFile_UT.Status.DeleteStep == FILE_DISABLED));
}

_SETUP_TEST(void) {
	TestState = 0;
	ArrangeSubState = 0;
	ActSubState = 0;
	AssertSubState = 0;
	FileNumber = 0;
	cycleCount = 0;
	NameMatch = 0;
	InNewLocation = 0;
	InOldLocation = 0;
	MultiSelectDirCopy = 0;
	MultiSelectFileCopy = 0;
	HmiFile.Status.SelectedIndex = 0;
	MpFileManagerUIConnect.File.Copy = 0;
	MpFileManagerUIConnect.File.CreateFolder = 0;
	MpFileManagerUIConnect.File.Cut = 0;
	MpFileManagerUIConnect.File.Delete = 0;
	MpFileManagerUIConnect.File.EnterFolder = 0;
	MpFileManagerUIConnect.File.FolderUp = 0;
	MpFileManagerUIConnect.File.MultiSelect = 0;
	MpFileManagerUIConnect.File.Paste = 0;
	MpFileManagerUIConnect.File.Refresh = 0;
	MpFileManagerUIConnect.File.Rename = 0;

	HmiFile_UT.Parameters.Fifo.Enable = false;
	HmiFile_UT.Parameters.Fifo.ScanInterval = 60;
	strcpy(HmiFile_UT.Parameters.Fifo.DeviceName, "mappUserXFiles");

	switch (SetupState)
	{
		case 0:
			TEST_BUSY_CONDITION(HmiFile_UT.Status.DeleteStep != FILE_DISABLED);
			for (USINT i=0; i<sizeof(HmiFile_UT.Status.FifoSelect)/sizeof(HmiFile_UT.Status.FifoSelect[0]); i++)
			{
				TEST_BUSY_CONDITION(HmiFile_UT.Status.FifoSelect[i] != 0);
			}

			DirInfo_UT.enable = true;
			DirInfo_UT.pDevice = (UDINT)&"mappUserXFiles";
			DirInfo_UT.pPath = (UDINT)&"";
			DirInfo(&DirInfo_UT);
			TEST_BUSY_CONDITION(DirInfo_UT.status == 65535);
			TEST_ABORT_CONDITION(DirInfo_UT.status != 0);
			NumberOfFiles = DirInfo_UT.filenum;
			CurrentFile = 0;
			SetupState = (NumberOfFiles == 0) ? 100 : 1;
			break;

		case 1:
			DirRead_UT.enable = true;
			DirRead_UT.pDevice = DirInfo_UT.pDevice;
			DirRead_UT.entry = 0;
			DirRead_UT.option = fiFILE;
			DirRead_UT.pData = (UDINT)&fileInfo;
			DirRead_UT.data_len = sizeof(fileInfo);
			DirRead(&DirRead_UT);
			TEST_BUSY_CONDITION(DirRead_UT.status == 65535);
			TEST_ABORT_CONDITION(DirRead_UT.status != 0);
			SetupState = 2;
			break;

		case 2:
			FileDelete_UT.enable = true;
			FileDelete_UT.pDevice = DirInfo_UT.pDevice;
			FileDelete_UT.pName = (UDINT)&fileInfo.Filename;
			FileDelete(&FileDelete_UT);
			TEST_BUSY_CONDITION(FileDelete_UT.status == 65535);
			TEST_ABORT_CONDITION(FileDelete_UT.status != 0);

			CurrentFile++;
			SetupState = (CurrentFile >= NumberOfFiles) ? 100 : 1;
			break;

		case 10:
			TEST_BUSY_CONDITION(MpFileManagerUIConnect_FIFO.Status == mpFILE_UI_STATUS_IDLE);
			MpFileManagerUIConnect_FIFO.File.Refresh = true;
			TEST_BUSY_CONDITION(MpFileManagerUIConnect_FIFO.Status == mpFILE_UI_STATUS_IDLE);
			MpFileManagerUIConnect_FIFO.File.Refresh = false;
			SetupState = 11;
			break;

		case 11:
			TEST_BUSY_CONDITION(MpFileManagerUIConnect_FIFO.Status != mpFILE_UI_STATUS_IDLE);
			SetupState = 100;
			break;

		case 100:
			TEST_DONE;
	}
	TEST_BUSY;
}

_TEARDOWN_TEST(void)
{
	HmiFile_UT.Parameters.Fifo.Enable = false;
	HmiFile_UT.Parameters.Fifo.ScanInterval = 60;

	TestState = 0;
	ArrangeSubState = 0;
	ActSubState = 0;
	AssertSubState = 0;
	cycleCount = 0;
	NameMatch = 0;
	InNewLocation = 0;
	InOldLocation = 0;
	MultiSelectDirCopy = 0;
	MultiSelectFileCopy = 0;
	HmiFile.Status.SelectedIndex = 0;
	MpFileManagerUIConnect.File.Copy = 0;
	MpFileManagerUIConnect.File.CreateFolder = 0;
	MpFileManagerUIConnect.File.Cut = 0;
	MpFileManagerUIConnect.File.Delete = 0;
	MpFileManagerUIConnect.File.EnterFolder = 0;
	MpFileManagerUIConnect.File.FolderUp = 0;
	MpFileManagerUIConnect.File.MultiSelect = 0;
	MpFileManagerUIConnect.File.Paste = 0;
	MpFileManagerUIConnect.File.Refresh = 0;
	MpFileManagerUIConnect.File.Rename = 0;
	brsmemcpy((UDINT)&MpFileManagerUIConnect.File.Filter, (UDINT)&"", sizeof(MpFileManagerUIConnect.File.Filter));

	HmiFile.Commands.Delete = 0;
	HmiFile.Commands.EnterFolder = 0;
	HmiFile.Commands.FolderUp = 0;
	HmiFile.Status.SelectedIndex = 0;

	FileCreate_0.enable = 0;
	FileClose_0.enable = 0;
	FileCreate(&FileCreate_0);
	FileClose(&FileClose_0);

	TEST_DONE;
}

_CYCLIC_SET(void)
{
	cycleCount++;
}

_TEST Create_Directory(void)
{
	TIMEOUT_TEST_CASE;

	switch (TestState)
	{
		case 0:
			// Select Recipe file device and input directory name
			switch (ArrangeSubState)
			{
				case 0:
					MpFileManagerUIConnect.DeviceList.SelectedIndex = 0;
					brsmemcpy((UDINT)&MpFileManagerUIConnect.File.NewName, (UDINT)&DirName, sizeof(MpFileManagerUIConnect.File.NewName));
					ArrangeSubState = 1;
					break;

				case 1:
					MpFileManagerUIConnect.File.Refresh = 1;
					ArrangeSubState = 2;
					break;

				case 2:
					TEST_BUSY_CONDITION(MpFileManagerUIConnect.Status != 0);
					MpFileManagerUIConnect.File.Refresh = 0;
					ArrangeSubState = 3;
					break;

				case 3:
					TEST_BUSY_CONDITION(MpFileManagerUIConnect.Status != 0);
					for(int i = 0; i < sizeof(MpFileManagerUIConnect.File.List.Items)/sizeof(MpFileManagerUIConnect.File.List.Items[0]); i++)
					{
						if(brsstrcmp((UDINT)&MpFileManagerUIConnect.File.List.Items[i].Name, (UDINT)&DirName) == 0)
						{
							TEST_ABORT_MSG("Directory with chosen name already exists");
						}
					}
					TestState = 1;
					break;
			}
			break;

		case 1:
			// Create directory
			switch (ActSubState)
			{
				case 0:
					MpFileManagerUIConnect.File.CreateFolder = 1;
					ActSubState = 1;
					break;

				case 1:
					TEST_BUSY_CONDITION(MpFileManagerUIConnect.Status != mpFILE_UI_STATUS_CREATE);
					MpFileManagerUIConnect.File.CreateFolder = 0;
					ActSubState = 2;

				case 2:
					TEST_BUSY_CONDITION(MpFileManagerUIConnect.Status != mpFILE_UI_STATUS_IDLE);
					MpFileManagerUIConnect.File.Refresh = 1;
					ActSubState = 3;
					break;

				case 3:
					TEST_BUSY_CONDITION(MpFileManagerUIConnect.Status != mpFILE_UI_STATUS_REFRESH);
					MpFileManagerUIConnect.File.Refresh = 0;
					ActSubState = 4;
					break;

				case 4:
					TEST_BUSY_CONDITION(MpFileManagerUIConnect.Status != mpFILE_UI_STATUS_IDLE);
					for(int i = 0; i < sizeof(MpFileManagerUIConnect.File.List.Items)/sizeof(MpFileManagerUIConnect.File.List.Items[0]); i++)
					{
						if(brsstrcmp((UDINT)&MpFileManagerUIConnect.File.List.Items[i].Name, (UDINT)&DirName) == 0)
						{
							NameMatch = 1;
						}
					}
					TestState = 2;
					break;
			}
			break;

		case 2:
			// Check save location for directory
			TEST_ASSERT(NameMatch);
			TEST_DONE;
			break;
	}
	TEST_BUSY;
}

_TEST Add_File(void)
{
	TIMEOUT_TEST_CASE;

	FileCreate(&FileCreate_0);
	FileClose(&FileClose_0);

	switch (TestState)
	{
		case 0:
			// Select Recipe file device and input file name
			switch (ArrangeSubState)
			{
				case 0:
					FileCreate_0.pDevice = (UDINT)&"USER";
					FileCreate_0.pFile = (UDINT)&CreateFileName;
					ArrangeSubState = 1;
					break;

				case 1:
					MpFileManagerUIConnect.File.Refresh = 1;
					ArrangeSubState = 2;
					break;

				case 2:
					TEST_BUSY_CONDITION(MpFileManagerUIConnect.Status != mpFILE_UI_STATUS_IDLE);
					MpFileManagerUIConnect.File.Refresh = 0;
					ArrangeSubState = 3;
					break;

				case 3: // Check to make sure there isn't already a file by the specified name in the directory
					TEST_BUSY_CONDITION(MpFileManagerUIConnect.Status != 0);
					for(int i = 0; i < sizeof(MpFileManagerUIConnect.File.List.Items)/sizeof(MpFileManagerUIConnect.File.List.Items[0]); i++)
					{
						if(brsstrcmp((UDINT)&MpFileManagerUIConnect.File.List.Items[i].Name, (UDINT)&CreateFileName) == 0)
						{
							TEST_ABORT_MSG("File with chosen name already exists");
						}
					}
					TestState = 1;
					break;
			}
			break;

		case 1:
			// Create file
			switch (ActSubState)
			{
				case 0:
					FileCreate_0.enable = 1;
					ActSubState = 1;
					break;

				case 1:
					if((FileCreate_0.status != 0) && (FileCreate_0.status != 65535))
					{
						TEST_ABORT_MSG("FileCreate function block has an error");
					}
					TEST_BUSY_CONDITION(FileCreate_0.status != 0);
					FileClose_0.ident = FileCreate_0.ident;
					FileClose_0.enable = 1;
					FileCreate_0.enable = 0;
					ActSubState = 2;
					break;

				case 2:
					if((FileClose_0.status != 0) && (FileClose_0.status != 65535))
					{
						TEST_ABORT_MSG("FileClose function block has an error");
					}
					TEST_BUSY_CONDITION(FileClose_0.status != 0);
					FileClose_0.enable = 0;
					MpFileManagerUIConnect.File.Refresh = 1;
					ActSubState = 3;
					break;

				case 3:
					TEST_BUSY_CONDITION(MpFileManagerUIConnect.Status != mpFILE_UI_STATUS_REFRESH);
					MpFileManagerUIConnect.File.Refresh = 0;
					ActSubState = 4;
					break;

				case 4:
					TEST_BUSY_CONDITION(MpFileManagerUIConnect.Status != mpFILE_UI_STATUS_IDLE);
					ActSubState = 5;
					break;

				case 5:
					for(int i = 0; i < sizeof(MpFileManagerUIConnect.File.List.Items)/sizeof(MpFileManagerUIConnect.File.List.Items[0]); i++)
					{
						if(brsstrcmp((UDINT)&MpFileManagerUIConnect.File.List.Items[i].Name, (UDINT)&CreateFileName) == 0)
						{
							NameMatch = 1;
						}
					}
					TestState = 2;
					break;
			}
			break;

		case 2:
			// Check save location for file
			TEST_ASSERT(NameMatch);
			TEST_DONE;
			break;
	}
	TEST_BUSY;
}

_TEST Copy_File(void)
{
	TIMEOUT_TEST_CASE;

	switch (TestState)
	{
		case 0:
			// Select Recipe file device and input name of file to be copied
			switch (ArrangeSubState)
			{
				case 0:
					MpFileManagerUIConnect.DeviceList.SelectedIndex = 0;
					ArrangeSubState = 1;
					break;

				case 1:
					for(int i = 0; i < sizeof(MpFileManagerUIConnect.File.List.Items)/sizeof(MpFileManagerUIConnect.File.List.Items[0]); i++)
					{
						if(brsstrcmp((UDINT)&MpFileManagerUIConnect.File.List.Items[i].Name, (UDINT)&CreateFileName) == 0)
							HmiFile.Status.SelectedIndex = i;
					}
					TestState = 1;
					break;
			}
			break;

		case 1:
			// Copy/paste file
			switch (ActSubState)
			{
				case 0:
					MpFileManagerUIConnect.File.Copy = 1;
					ActSubState = 1;
					break;

				case 1:
					MpFileManagerUIConnect.File.Copy = 0;
					MpFileManagerUIConnect.File.Paste = 1;
					ActSubState = 2;
					break;

				case 2:
					MpFileManagerUIConnect.File.Paste = 0;
					TEST_BUSY_CONDITION(MpFileManagerUIConnect.Status != mpFILE_UI_STATUS_PASTE);
					ActSubState = 3;
					break;

				case 3:
					TEST_BUSY_CONDITION(MpFileManagerUIConnect.Status != mpFILE_UI_STATUS_IDLE);
					MpFileManagerUIConnect.File.Refresh = 1;
					ActSubState = 4;
					break;

				case 4:
					TEST_BUSY_CONDITION(MpFileManagerUIConnect.Status != mpFILE_UI_STATUS_REFRESH);
					MpFileManagerUIConnect.File.Refresh = 0;
					ActSubState = 5;
					break;

				case 5:
					// Check file list for copied file
					TEST_BUSY_CONDITION(MpFileManagerUIConnect.Status != mpFILE_UI_STATUS_IDLE);
					for(int i = 0; i < sizeof(MpFileManagerUIConnect.File.List.Items)/sizeof(MpFileManagerUIConnect.File.List.Items[0]); i++)
					{
						if(brsstrcmp((UDINT)&MpFileManagerUIConnect.File.List.Items[i].Name, (UDINT)&CopiedFileName) == 0)
						{
							NameMatch = 1;
						}
					}
					TestState = 2;
					break;
			}
			break;

		case 2:
			// Check if copied file was found
			TEST_ASSERT(NameMatch);
			TEST_DONE;
			break;
	}
	TEST_BUSY;
}

_TEST Copy_Directory(void)
{
	TIMEOUT_TEST_CASE;

	switch (TestState)
	{
		case 0:
			// Select Recipe file device and input name of directory to be copied
			switch (ArrangeSubState)
			{
				case 0:
					MpFileManagerUIConnect.DeviceList.SelectedIndex = 0;
					ArrangeSubState = 1;
					break;

				case 1:
					for(int i = 0; i < sizeof(MpFileManagerUIConnect.File.List.Items)/sizeof(MpFileManagerUIConnect.File.List.Items[0]); i++)
					{
						if(brsstrcmp((UDINT)&MpFileManagerUIConnect.File.List.Items[i].Name, (UDINT)&DirName) == 0)
							HmiFile.Status.SelectedIndex = i;
					}
					TestState = 1;
					break;
			}
			break;

		case 1:
			// Copy/paste directory
			switch (ActSubState)
			{
				case 0:
					MpFileManagerUIConnect.File.Copy = 1;
					ActSubState = 1;
					break;

				case 1:
					MpFileManagerUIConnect.File.Copy = 0;
					MpFileManagerUIConnect.File.Paste = 1;
					ActSubState = 2;
					break;

				case 2:
					MpFileManagerUIConnect.File.Paste = 0;
					TEST_BUSY_CONDITION(MpFileManagerUIConnect.Status != mpFILE_UI_STATUS_PASTE);
					ActSubState = 3;
					break;

				case 3:
					TEST_BUSY_CONDITION(MpFileManagerUIConnect.Status != mpFILE_UI_STATUS_IDLE);
					MpFileManagerUIConnect.File.Refresh = 1;
					ActSubState = 4;
					break;

				case 4:
					TEST_BUSY_CONDITION(MpFileManagerUIConnect.Status != mpFILE_UI_STATUS_REFRESH);
					MpFileManagerUIConnect.File.Refresh = 0;
					ActSubState = 5;
					break;

				case 5:
					// Check file list for copied directory
					TEST_BUSY_CONDITION(MpFileManagerUIConnect.Status != mpFILE_UI_STATUS_IDLE);
					for(int i = 0; i < sizeof(MpFileManagerUIConnect.File.List.Items)/sizeof(MpFileManagerUIConnect.File.List.Items[0]); i++)
					{
						if(brsstrcmp((UDINT)&MpFileManagerUIConnect.File.List.Items[i].Name, (UDINT)&CopiedDirName) == 0)
						{
							NameMatch = 1;
						}
					}
					TestState = 2;
					break;
			}
			break;

		case 2:
			// Check if copied directory was found
			TEST_ASSERT(NameMatch);
			TEST_DONE;
			break;
	}
	TEST_BUSY;
}

_TEST Rename_File(void)
{
	TIMEOUT_TEST_CASE;

	switch (TestState)
	{
		case 0:
			// Select Recipe file device and input name of file to be renamed and new name
			switch (ArrangeSubState)
			{
				case 0:
					MpFileManagerUIConnect.DeviceList.SelectedIndex = 0;
					brsmemcpy((UDINT)&MpFileManagerUIConnect.File.NewName, (UDINT)&NewFileName, sizeof(MpFileManagerUIConnect.File.NewName));
					ArrangeSubState = 1;
					break;

				case 1:
					for(int i = 0; i < sizeof(MpFileManagerUIConnect.File.List.Items)/sizeof(MpFileManagerUIConnect.File.List.Items[0]); i++)
					{
						if(brsstrcmp((UDINT)&MpFileManagerUIConnect.File.List.Items[i].Name, (UDINT)&CopiedFileName) == 0)
							HmiFile.Status.SelectedIndex = i;
					}
					TestState = 1;
					break;
			}
			break;

		case 1:
			// Rename file
			switch (ActSubState)
			{
				case 0:
					MpFileManagerUIConnect.File.Rename = 1;
					ActSubState = 1;
					break;

				case 1:
					MpFileManagerUIConnect.File.Rename = 0;
					TEST_BUSY_CONDITION(MpFileManagerUIConnect.Status != mpFILE_UI_STATUS_IDLE);
					MpFileManagerUIConnect.File.Refresh = 1;
					ActSubState = 2;
					break;

				case 2:
					TEST_BUSY_CONDITION(MpFileManagerUIConnect.Status != mpFILE_UI_STATUS_REFRESH);
					MpFileManagerUIConnect.File.Refresh = 0;
					ActSubState = 3;
					break;

				case 3:
					// Check file list for renamed file
					TEST_BUSY_CONDITION(MpFileManagerUIConnect.Status != mpFILE_UI_STATUS_IDLE);
					for(int i = 0; i < sizeof(MpFileManagerUIConnect.File.List.Items)/sizeof(MpFileManagerUIConnect.File.List.Items[0]); i++)
					{
						if(brsstrcmp((UDINT)&MpFileManagerUIConnect.File.List.Items[i].Name, (UDINT)&NewFileName) == 0)
						{
							NameMatch = 1;
						}
					}
					TestState = 2;
					break;
			}
			break;

		case 2:
			// Check if renamed file was found
			TEST_ASSERT(NameMatch);
			TEST_DONE;
			break;
	}
	TEST_BUSY;
}

_TEST Rename_Directory(void)
{
	TIMEOUT_TEST_CASE;

	switch (TestState)
	{
		case 0:
			// Select Recipe file device and input name of directory to be renamed and new name
			switch (ArrangeSubState)
			{
				case 0:
					MpFileManagerUIConnect.DeviceList.SelectedIndex = 0;
					brsmemcpy((UDINT)&MpFileManagerUIConnect.File.NewName, (UDINT)&NewDirName, sizeof(MpFileManagerUIConnect.File.NewName));
					ArrangeSubState = 1;
					break;

				case 1:
					for(int i = 0; i < sizeof(MpFileManagerUIConnect.File.List.Items)/sizeof(MpFileManagerUIConnect.File.List.Items[0]); i++)
					{
						if(brsstrcmp((UDINT)&MpFileManagerUIConnect.File.List.Items[i].Name, (UDINT)&CopiedDirName) == 0)
							HmiFile.Status.SelectedIndex = i;
					}
					TestState = 1;
					break;
			}
			break;

		case 1:
			// Rename directory
			switch (ActSubState)
			{
				case 0:
					MpFileManagerUIConnect.File.Rename = 1;
					ActSubState = 1;
					break;

				case 1:
					MpFileManagerUIConnect.File.Rename = 0;
					TEST_BUSY_CONDITION(MpFileManagerUIConnect.Status != mpFILE_UI_STATUS_IDLE);
					MpFileManagerUIConnect.File.Refresh = 1;
					ActSubState = 2;
					break;

				case 2:
					TEST_BUSY_CONDITION(MpFileManagerUIConnect.Status != mpFILE_UI_STATUS_REFRESH);
					MpFileManagerUIConnect.File.Refresh = 0;
					ActSubState = 3;
					break;

				case 3:
					// Check file list for renamed directory
					TEST_BUSY_CONDITION(MpFileManagerUIConnect.Status != mpFILE_UI_STATUS_IDLE);
					for(int i = 0; i < sizeof(MpFileManagerUIConnect.File.List.Items)/sizeof(MpFileManagerUIConnect.File.List.Items[0]); i++)
					{
						if(brsstrcmp((UDINT)&MpFileManagerUIConnect.File.List.Items[i].Name, (UDINT)&NewDirName) == 0)
						{
							NameMatch = 1;
						}
					}
					TestState = 2;
					break;
			}
			break;

		case 2:
			// Check if renamed directory was found
			TEST_ASSERT(NameMatch);
			TEST_DONE;
			break;
	}
	TEST_BUSY;
}

_TEST Cut_Paste_File(void)
{
	TIMEOUT_TEST_CASE;

	switch (TestState)
	{
		case 0:
			// Select Recipe file device and input name of file to be cut
			switch (ArrangeSubState)
			{
				case 0:
					MpFileManagerUIConnect.DeviceList.SelectedIndex = 0;
					MpFileManagerUIConnect.File.Refresh = 1;
					ArrangeSubState = 1;
					break;

			case 1:
					TEST_BUSY_CONDITION(MpFileManagerUIConnect.Status != mpFILE_UI_STATUS_REFRESH);
					MpFileManagerUIConnect.File.Refresh = 0;
					ArrangeSubState = 2;
					break;

				case 2:
					TEST_BUSY_CONDITION(MpFileManagerUIConnect.Status != mpFILE_UI_STATUS_IDLE);
					for(int i = 0; i < sizeof(MpFileManagerUIConnect.File.List.Items)/sizeof(MpFileManagerUIConnect.File.List.Items[0]); i++)
					{
						if(brsstrcmp((UDINT)&MpFileManagerUIConnect.File.List.Items[i].Name, (UDINT)&NewFileName) == 0)
							HmiFile.Status.SelectedIndex = i;
					}
					TestState = 1;
					break;
			}
			break;

		case 1:
			// Cut/paste file
			switch (ActSubState)
			{
				case 0:
					MpFileManagerUIConnect.File.Cut = 1;
					ActSubState = 1;
					break;

				case 1:
					MpFileManagerUIConnect.File.Cut = 0;
					for(int i = 0; i < sizeof(MpFileManagerUIConnect.File.List.Items)/sizeof(MpFileManagerUIConnect.File.List.Items[0]); i++)
					{
						if(brsstrcmp((UDINT)&MpFileManagerUIConnect.File.List.Items[i].Name, (UDINT)&DirName) == 0)
							HmiFile.Status.SelectedIndex = i;
					}
					ActSubState = 2;
					break;

				case 2:
					HmiFile.Commands.EnterFolder = 1;
					TEST_BUSY_CONDITION(MpFileManagerUIConnect.Status != mpFILE_UI_STATUS_CHANGE_DIR);
					HmiFile.Commands.EnterFolder = 0;
					ActSubState = 3;
					break;

				case 3:
					TEST_BUSY_CONDITION(MpFileManagerUIConnect.Status != mpFILE_UI_STATUS_IDLE);
					MpFileManagerUIConnect.File.Paste = 1;
					ActSubState = 4;
					break;

				case 4:
					MpFileManagerUIConnect.File.Paste = 0;
					TEST_BUSY_CONDITION(MpFileManagerUIConnect.Status != mpFILE_UI_STATUS_PASTE);
					ActSubState = 5;
					break;

				case 5:
					TEST_BUSY_CONDITION(MpFileManagerUIConnect.Status != mpFILE_UI_STATUS_IDLE);
					MpFileManagerUIConnect.File.Refresh = 1;
					ActSubState = 6;
					break;

				case 6:
					TEST_BUSY_CONDITION(MpFileManagerUIConnect.Status != mpFILE_UI_STATUS_REFRESH);
					MpFileManagerUIConnect.File.Refresh = 0;
					ActSubState = 7;
					break;

				case 7:
					// Check paste location for cut file
					TEST_BUSY_CONDITION(MpFileManagerUIConnect.Status != mpFILE_UI_STATUS_IDLE);
					for(int i = 0; i < sizeof(MpFileManagerUIConnect.File.List.Items)/sizeof(MpFileManagerUIConnect.File.List.Items[0]); i++)
					{
						if(brsstrcmp((UDINT)&MpFileManagerUIConnect.File.List.Items[i].Name, (UDINT)&NewFileName) == 0)
						{
							InNewLocation = 1;
						}
					}
					HmiFile.Commands.FolderUp = 1;
					ActSubState = 8;
					break;

				case 8:
					TEST_BUSY_CONDITION(MpFileManagerUIConnect.Status != mpFILE_UI_STATUS_CHANGE_DIR);
					HmiFile.Commands.FolderUp = 0;
					ActSubState = 9;
					break;

				case 9:
					// Check old location for cut file
					TEST_BUSY_CONDITION(MpFileManagerUIConnect.Status != mpFILE_UI_STATUS_IDLE);
					for(int i = 0; i < sizeof(MpFileManagerUIConnect.File.List.Items)/sizeof(MpFileManagerUIConnect.File.List.Items[0]); i++)
					{
						if(brsstrcmp((UDINT)&MpFileManagerUIConnect.File.List.Items[i].Name, (UDINT)&NewFileName) == 0)
						{
							InOldLocation = 1;
						}
					}
					TestState = 2;
					break;
			}
			break;

		case 2:
			// Check new and old locations for file
			TEST_ASSERT(InNewLocation);
			TEST_ASSERT(!InOldLocation);
			TEST_DONE;
			break;
	}
	TEST_BUSY;
}

_TEST Cut_Paste_Directory(void)
{
	TIMEOUT_TEST_CASE;

	switch (TestState)
	{
		case 0:
			// Select Recipe file device and input name of directory to be cut
			switch (ArrangeSubState)
			{
				case 0:
					MpFileManagerUIConnect.DeviceList.SelectedIndex = 0;
					ArrangeSubState = 1;
					break;

				case 1:
					for(int i = 0; i < sizeof(MpFileManagerUIConnect.File.List.Items)/sizeof(MpFileManagerUIConnect.File.List.Items[0]); i++)
					{
						if(brsstrcmp((UDINT)&MpFileManagerUIConnect.File.List.Items[i].Name, (UDINT)&NewDirName) == 0)
							HmiFile.Status.SelectedIndex = i;
					}
					TestState = 1;
					break;
			}
			break;

		case 1:
			// Cut/paste directory
			switch (ActSubState)
			{
				case 0:
					MpFileManagerUIConnect.File.Cut = 1;
					ActSubState = 1;
					break;

				case 1:
					MpFileManagerUIConnect.File.Cut = 0;
					MpFileManagerUIConnect.File.Refresh = 1;
					ActSubState = 2;
					break;

				case 2:
					TEST_BUSY_CONDITION(MpFileManagerUIConnect.Status != mpFILE_UI_STATUS_REFRESH);
					MpFileManagerUIConnect.File.Refresh = 0;
					ActSubState = 3;
					break;

				case 3:
					// Find folder to paste directory into
					TEST_BUSY_CONDITION(MpFileManagerUIConnect.Status != mpFILE_UI_STATUS_IDLE);
					for(int i = 0; i < sizeof(MpFileManagerUIConnect.File.List.Items)/sizeof(MpFileManagerUIConnect.File.List.Items[0]); i++)
					{
						if(brsstrcmp((UDINT)&MpFileManagerUIConnect.File.List.Items[i].Name, (UDINT)&DirName) == 0)
							HmiFile.Status.SelectedIndex = i;
					}
					ActSubState = 4;
					break;

				case 4:
					MpFileManagerUIConnect.File.Refresh = 1;
					ActSubState = 5;
					break;

				case 5:
					TEST_BUSY_CONDITION(MpFileManagerUIConnect.Status != mpFILE_UI_STATUS_REFRESH);
					MpFileManagerUIConnect.File.Refresh = 0;
					ActSubState = 6;
					break;

				case 6:
					TEST_BUSY_CONDITION(MpFileManagerUIConnect.Status != mpFILE_UI_STATUS_IDLE);
					HmiFile.Commands.EnterFolder = 1;
					ActSubState = 7;
					break;

				case 7:
					HmiFile.Commands.EnterFolder = 0;
					TEST_BUSY_CONDITION(MpFileManagerUIConnect.Status != mpFILE_UI_STATUS_CHANGE_DIR);
					ActSubState = 8;
					break;

				case 8:
					TEST_BUSY_CONDITION(MpFileManagerUIConnect.Status != mpFILE_UI_STATUS_IDLE);
					MpFileManagerUIConnect.File.Paste = 1;
					ActSubState = 9;
					break;

				case 9:
					MpFileManagerUIConnect.File.Paste = 0;
					TEST_BUSY_CONDITION(MpFileManagerUIConnect.Status != mpFILE_UI_STATUS_PASTE);
					ActSubState = 10;
					break;

				case 10:
					TEST_BUSY_CONDITION(MpFileManagerUIConnect.Status != mpFILE_UI_STATUS_IDLE);
					MpFileManagerUIConnect.File.Refresh = 1;
					ActSubState = 11;
					break;

				case 11:
					TEST_BUSY_CONDITION(MpFileManagerUIConnect.Status != mpFILE_UI_STATUS_REFRESH);
					MpFileManagerUIConnect.File.Refresh = 0;
					ActSubState = 12;
					break;

				case 12:
					// Check new location for cut directory
					TEST_BUSY_CONDITION(MpFileManagerUIConnect.Status != mpFILE_UI_STATUS_IDLE);
					for(int i = 0; i < sizeof(MpFileManagerUIConnect.File.List.Items)/sizeof(MpFileManagerUIConnect.File.List.Items[0]); i++)
					{
						if(brsstrcmp((UDINT)&MpFileManagerUIConnect.File.List.Items[i].Name, (UDINT)&NewDirName) == 0)
						{
							InNewLocation = 1;
						}
					}
					HmiFile.Commands.FolderUp = 1;
					ActSubState = 13;
					break;

				case 13:
					TEST_BUSY_CONDITION(MpFileManagerUIConnect.Status != mpFILE_UI_STATUS_CHANGE_DIR);
					HmiFile.Commands.FolderUp = 0;
					ActSubState = 14;
					break;

				case 14:
					// Check old location for cut directory
					TEST_BUSY_CONDITION(MpFileManagerUIConnect.Status != mpFILE_UI_STATUS_IDLE);
					for(int i = 0; i < sizeof(MpFileManagerUIConnect.File.List.Items)/sizeof(MpFileManagerUIConnect.File.List.Items[0]); i++)
					{
						if(brsstrcmp((UDINT)&MpFileManagerUIConnect.File.List.Items[i].Name, (UDINT)&NewDirName) == 0)
						{
							InOldLocation = 1;
						}
					}
					TestState = 2;
					break;
			}
			break;

		case 2:
			// Check new and old locations for directory
			TEST_ASSERT(InNewLocation);
			TEST_ASSERT(!InOldLocation);
			TEST_DONE;
			break;
	}
	TEST_BUSY;
}

_TEST Multiselect(void)
{
	TIMEOUT_TEST_CASE;

	switch (TestState)
	{
		case 0:
			// Select Recipe file device and navigate into directory with test files
			switch (ArrangeSubState)
			{
				case 0:
					MpFileManagerUIConnect.DeviceList.SelectedIndex = 0;
					ArrangeSubState = 1;
					break;

				case 1:
					for(int i = 0; i < sizeof(MpFileManagerUIConnect.File.List.Items)/sizeof(MpFileManagerUIConnect.File.List.Items[0]); i++)
					{
						if(brsstrcmp((UDINT)&MpFileManagerUIConnect.File.List.Items[i].Name, (UDINT)&DirName) == 0)
							HmiFile.Status.SelectedIndex = i;
					}
					ArrangeSubState = 2;
					break;

			case 2:
					MpFileManagerUIConnect.File.Refresh = 1;
					TEST_BUSY_CONDITION(MpFileManagerUIConnect.Status != mpFILE_UI_STATUS_REFRESH);
					MpFileManagerUIConnect.File.Refresh = 0;
					ArrangeSubState = 3;
					break;

			case 3:
					TEST_BUSY_CONDITION(MpFileManagerUIConnect.Status != mpFILE_UI_STATUS_IDLE);
					HmiFile.Commands.EnterFolder = 1;
					ArrangeSubState = 4;
					break;

				case 4:
					HmiFile.Commands.EnterFolder = 0;
					TEST_BUSY_CONDITION(MpFileManagerUIConnect.Status != mpFILE_UI_STATUS_CHANGE_DIR);
					ArrangeSubState = 5;
					break;

				case 5:
					TEST_BUSY_CONDITION(MpFileManagerUIConnect.Status != mpFILE_UI_STATUS_IDLE);
					TestState = 1;
					break;
			}
			break;

		case 1:
			// Select multiple files/directories and copy/paste
			switch (ActSubState)
			{
				case 0:
					MpFileManagerUIConnect.File.MultiSelect = 1;
					ActSubState = 1;
					break;

				case 1:
					MpFileManagerUIConnect.File.List.Items[0].IsSelected = 1;
					MpFileManagerUIConnect.File.List.Items[1].IsSelected = 1;
					ActSubState = 2;
					break;

				case 2:
					MpFileManagerUIConnect.File.Copy = 1;
					ActSubState = 3;
					break;

				case 3:
					MpFileManagerUIConnect.File.Copy = 0;
					MpFileManagerUIConnect.File.MultiSelect = 0;
					MpFileManagerUIConnect.File.Paste = 1;
					ActSubState = 4;
					break;

				case 4:
					TEST_BUSY_CONDITION(MpFileManagerUIConnect.Status != mpFILE_UI_STATUS_PASTE);
					MpFileManagerUIConnect.File.Paste = 0;
					ActSubState = 5;
					break;

				case 5:
					TEST_BUSY_CONDITION(MpFileManagerUIConnect.Status != mpFILE_UI_STATUS_IDLE);
					MpFileManagerUIConnect.File.Refresh = 1;
					ActSubState = 6;
					break;

				case 6:
					TEST_BUSY_CONDITION(MpFileManagerUIConnect.Status != mpFILE_UI_STATUS_REFRESH);
					MpFileManagerUIConnect.File.Refresh = 0;
					ActSubState = 7;
					break;

				case 7:
					// Check for copied file
					TEST_BUSY_CONDITION(MpFileManagerUIConnect.Status != mpFILE_UI_STATUS_IDLE);
					for(int i = 0; i < sizeof(MpFileManagerUIConnect.File.List.Items)/sizeof(MpFileManagerUIConnect.File.List.Items[0]); i++)
					{
						if(brsstrcmp((UDINT)&MpFileManagerUIConnect.File.List.Items[i].Name, (UDINT)&CopiedNewFileName) == 0)
							MultiSelectFileCopy = 1;
					}
					ActSubState = 8;
					break;

				case 8:
					// Check for copied directory
					for(int i = 0; i < sizeof(MpFileManagerUIConnect.File.List.Items)/sizeof(MpFileManagerUIConnect.File.List.Items[0]); i++)
					{
						if(brsstrcmp((UDINT)&MpFileManagerUIConnect.File.List.Items[i].Name, (UDINT)&CopiedNewDirName) == 0)
							MultiSelectDirCopy = 1;
					}
					ActSubState = 9;
					break;

				case 9:
					HmiFile.Commands.FolderUp = 1;
					TEST_BUSY_CONDITION(MpFileManagerUIConnect.Status != mpFILE_UI_STATUS_CHANGE_DIR);
					HmiFile.Commands.FolderUp = 0;
					ActSubState = 10;
					break;

				case 10:
					TEST_BUSY_CONDITION(MpFileManagerUIConnect.Status != mpFILE_UI_STATUS_IDLE);
					TestState = 2;
					break;
			}
			break;

		case 2:
			// Check if copied file and directory were found
			TEST_ASSERT(MultiSelectFileCopy);
			TEST_ASSERT(MultiSelectDirCopy);
			TEST_DONE;
			break;
	}
	TEST_BUSY;
}

_TEST Search(void)
{
	TIMEOUT_TEST_CASE;

	switch (TestState)
	{
		case 0:
			// Set filter value to name of file
			MpFileManagerUIConnect.DeviceList.SelectedIndex = 0;
			brsmemcpy((UDINT)&MpFileManagerUIConnect.File.Filter, (UDINT)&CreateFileName, sizeof(MpFileManagerUIConnect.File.Filter));
			TestState = 1;
			break;

		case 1:
			// Refresh MpFileManagerUIConnect
			switch (ActSubState)
			{
				case 0:
					MpFileManagerUIConnect.File.Refresh = 1;
					ActSubState = 1;
					break;

				case 1:
					TEST_BUSY_CONDITION(MpFileManagerUIConnect.Status != mpFILE_UI_STATUS_REFRESH);
					MpFileManagerUIConnect.File.Refresh = 0;
					ActSubState = 2;
					break;

				case 2:
					// Check if the first item in the file list is the desired file
					TEST_BUSY_CONDITION(MpFileManagerUIConnect.Status != mpFILE_UI_STATUS_IDLE);
					if(brsstrcmp((UDINT)&MpFileManagerUIConnect.File.List.Items[0].Name, (UDINT)&CreateFileName) == 0)
						NameMatch = 1;
					ActSubState = 3;
					break;

				case 3:
					// Reset filter
					brsmemcpy((UDINT)&MpFileManagerUIConnect.File.Filter, (UDINT)&"", sizeof(MpFileManagerUIConnect.File.Filter));
					MpFileManagerUIConnect.File.Refresh = 1;
					ActSubState = 4;
					break;

				case 4:
					TEST_BUSY_CONDITION(MpFileManagerUIConnect.Status != mpFILE_UI_STATUS_REFRESH);
					MpFileManagerUIConnect.File.Refresh = 0;
					ActSubState = 5;
					break;

				case 5:
					TEST_BUSY_CONDITION(MpFileManagerUIConnect.Status != mpFILE_UI_STATUS_IDLE);
					TestState = 2;
					break;
			}
			break;

		case 2:
			// Check if filter worked
			TEST_ASSERT(NameMatch);
			TEST_DONE;
			break;
	}
	TEST_BUSY;
}

_TEST Enter_Folder(void)
{
	TIMEOUT_TEST_CASE;

	switch (TestState)
	{
		case 0:
			// Select folder to enter
			for(int i = 0; i < sizeof(MpFileManagerUIConnect.File.List.Items)/sizeof(MpFileManagerUIConnect.File.List.Items[0]); i++)
			{
				if(brsstrcmp((UDINT)&MpFileManagerUIConnect.File.List.Items[i].Name, (UDINT)&DirName) == 0)
					HmiFile.Status.SelectedIndex = i;
			}
			TestState = 1;
			break;

		case 1:
			// Give HMI command to enter folder
			switch (ActSubState)
			{
				case 0:
					// Acts as a delay to let the folder selection make its way to FileMgr task
					ActSubState = 1;
					break;

				case 1:
					HmiFile.Commands.EnterFolder = 1;
					ActSubState = 2;
					break;

				case 2:
					HmiFile.Commands.EnterFolder = 0;
					TEST_BUSY_CONDITION(MpFileManagerUIConnect.Status != mpFILE_UI_STATUS_CHANGE_DIR);
					ActSubState = 3;
					break;

				case 3:
					// Check if current directory matches what is expected
					TEST_BUSY_CONDITION(MpFileManagerUIConnect.Status != mpFILE_UI_STATUS_IDLE);
					if(brsstrcmp((UDINT)&MpFileManagerUIConnect.File.PathInfo.CurrentDir , (UDINT)&DirName) == 0)
						NameMatch = 1;
					ActSubState = 4;
					break;

				case 4:
					// Go back up to root folder
					HmiFile.Commands.FolderUp = 1;
					ActSubState = 5;
					break;

				case 5:
					TEST_BUSY_CONDITION(MpFileManagerUIConnect.Status != mpFILE_UI_STATUS_CHANGE_DIR);
					HmiFile.Commands.FolderUp = 0;
					ActSubState = 6;
					break;

				case 6:
					TEST_BUSY_CONDITION(MpFileManagerUIConnect.Status != mpFILE_UI_STATUS_IDLE);
					TestState = 2;
					break;
			}
			break;

		case 2:
			TEST_ASSERT(NameMatch);
			TEST_DONE;
			break;
	}
	TEST_BUSY;
}

_TEST Go_Up_Level(void)
{
	TIMEOUT_TEST_CASE;

	switch (TestState)
	{
		case 0:
			// Select folder to enter
			for(int i = 0; i < sizeof(MpFileManagerUIConnect.File.List.Items)/sizeof(MpFileManagerUIConnect.File.List.Items[0]); i++)
			{
				if(brsstrcmp((UDINT)&MpFileManagerUIConnect.File.List.Items[i].Name, (UDINT)&DirName) == 0)
					HmiFile.Status.SelectedIndex = i;
			}
			TestState = 1;
			break;

		case 1:
			// Give HMI command to enter folder
			switch (ActSubState)
			{
				case 0:
					// Acts as a delay to let the folder selection make its way to FileMgr task
					ActSubState = 1;
					break;

				case 1:
					HmiFile.Commands.EnterFolder = 1;
					ActSubState = 2;
					break;

				case 2:
					HmiFile.Commands.EnterFolder = 0;
					TEST_BUSY_CONDITION(MpFileManagerUIConnect.Status != mpFILE_UI_STATUS_CHANGE_DIR);
					ActSubState = 3;
					break;

				case 3:
					// Check if folder was successfully entered
					TEST_BUSY_CONDITION(MpFileManagerUIConnect.Status != mpFILE_UI_STATUS_IDLE);
					if(brsstrcmp((UDINT)&MpFileManagerUIConnect.File.PathInfo.CurrentDir , (UDINT)&DirName) != 0)
					{
						TEST_ABORT_MSG("Directory was not successfully entered");
					}
					ActSubState = 4;
					break;

				case 4:
					// Go back up to root folder
					HmiFile.Commands.FolderUp = 1;
					ActSubState = 5;
					break;

				case 5:
					TEST_BUSY_CONDITION(MpFileManagerUIConnect.Status != mpFILE_UI_STATUS_CHANGE_DIR);
					HmiFile.Commands.FolderUp = 0;
					ActSubState = 6;
					break;

				case 6:
					// Check if folder level went back up to the root
					TEST_BUSY_CONDITION(MpFileManagerUIConnect.Status != mpFILE_UI_STATUS_IDLE);
					if(brsstrcmp((UDINT)&MpFileManagerUIConnect.File.PathInfo.CurrentDir , (UDINT)&"") == 0)
						NameMatch = 1;
					TestState = 2;
					break;
			}
			break;

		case 2:
			TEST_ASSERT(NameMatch);
			TEST_DONE;
			break;
	}
	TEST_BUSY;
}

_TEST Change_Sort(void)
{
	TIMEOUT_TEST_CASE;

	switch (TestState)
	{
		case 0:
			// Change SortOrder value
			MpFileManagerUIConnect.File.SortOrder = 5;
			TestState = 1;
			break;

		case 1:
			switch (ActSubState)
			{
				case 0:
					// Wait for sort to take effect
					TEST_BUSY_CONDITION(MpFileManagerUIConnect.Status != mpFILE_UI_STATUS_SORT);
					ActSubState = 1;
					break;

				case 1:
					// Make sure sort worked correctly
					TEST_BUSY_CONDITION(MpFileManagerUIConnect.Status != mpFILE_UI_STATUS_IDLE);
					if(brsstrcmp((UDINT)&MpFileManagerUIConnect.File.List.Items[0].Name, (UDINT)&DirName) == 0)
						NameMatch = 1;
					ActSubState = 2;
					break;

				case 2:
					MpFileManagerUIConnect.File.SortOrder = 0;
					TEST_BUSY_CONDITION(MpFileManagerUIConnect.Status != mpFILE_UI_STATUS_SORT);
					ActSubState = 3;
					break;

				case 3:
					TEST_BUSY_CONDITION(MpFileManagerUIConnect.Status != mpFILE_UI_STATUS_IDLE);
					TestState = 2;
					break;
			}
			break;

		case 2:
			TEST_ASSERT(NameMatch);
			TEST_DONE;
			break;
	}
	TEST_BUSY;
}

_TEST Delete_File(void)
{
	TIMEOUT_TEST_CASE;

	switch (TestState)
	{
		case 0:
			// Select file to be deleted
			for(int i = 0; i < sizeof(MpFileManagerUIConnect.File.List.Items)/sizeof(MpFileManagerUIConnect.File.List.Items[0]); i++)
			{
				if(brsstrcmp((UDINT)&MpFileManagerUIConnect.File.List.Items[i].Name, (UDINT)&CreateFileName) == 0)
					HmiFile.Status.SelectedIndex = i;
			}
			TestState = 1;
			break;

		case 1:
			// Delete file
			switch (ActSubState)
			{
				case 0:
					MpFileManagerUIConnect.File.Delete = 1;
					TEST_BUSY_CONDITION(MpFileManagerUIConnect.Status != mpFILE_UI_STATUS_DELETE);
					MpFileManagerUIConnect.File.Delete = 0;
					ActSubState = 1;
					break;

				case 1:
					MpFileManagerUIConnect.MessageBox.Confirm = 1;
					TEST_BUSY_CONDITION(MpFileManagerUIConnect.Status != mpFILE_UI_STATUS_IDLE);
					MpFileManagerUIConnect.MessageBox.Confirm = 0;
					ActSubState = 2;
					break;

				case 2:
					MpFileManagerUIConnect.File.Refresh = 1;
					ActSubState = 3;
					break;

				case 3:
					TEST_BUSY_CONDITION(MpFileManagerUIConnect.Status != mpFILE_UI_STATUS_REFRESH);
					MpFileManagerUIConnect.File.Refresh = 0;
					ActSubState = 4;
					break;

				case 4:
					// Check for file
					TEST_BUSY_CONDITION(MpFileManagerUIConnect.Status != mpFILE_UI_STATUS_IDLE);
					for(int i = 0; i < sizeof(MpFileManagerUIConnect.File.List.Items)/sizeof(MpFileManagerUIConnect.File.List.Items[0]); i++)
					{
						if(brsstrcmp((UDINT)&MpFileManagerUIConnect.File.List.Items[i].Name, (UDINT)&CreateFileName) == 0)
							NameMatch = 1;
					}
					TestState = 2;
					break;
			}
			break;

		case 2:
			// Check if file was deleted
			TEST_ASSERT(!NameMatch);
			TEST_DONE;
			break;
	}
	TEST_BUSY;
}

_TEST Delete_Directory(void)
{
	TIMEOUT_TEST_CASE;

	switch (TestState)
	{
		case 0:
			// Select directory to be deleted
			for(int i = 0; i < sizeof(MpFileManagerUIConnect.File.List.Items)/sizeof(MpFileManagerUIConnect.File.List.Items[0]); i++)
			{
				if(brsstrcmp((UDINT)&MpFileManagerUIConnect.File.List.Items[i].Name, (UDINT)&DirName) == 0)
					HmiFile.Status.SelectedIndex = i;
			}
			TestState = 1;
			break;

		case 1:
			// Delete file
			switch (ActSubState)
			{
				case 0:
					MpFileManagerUIConnect.File.Delete = 1;
					TEST_BUSY_CONDITION(MpFileManagerUIConnect.Status != mpFILE_UI_STATUS_DELETE);
					MpFileManagerUIConnect.File.Delete = 0;
					ActSubState = 1;
					break;

				case 1:
					MpFileManagerUIConnect.MessageBox.Confirm = 1;
					TEST_BUSY_CONDITION(MpFileManagerUIConnect.Status != mpFILE_UI_STATUS_IDLE);
					MpFileManagerUIConnect.MessageBox.Confirm = 0;
					ActSubState = 2;
					break;
					break;

				case 2:
					MpFileManagerUIConnect.File.Refresh = 1;
					ActSubState = 3;
					break;

				case 3:
					TEST_BUSY_CONDITION(MpFileManagerUIConnect.Status != mpFILE_UI_STATUS_REFRESH);
					MpFileManagerUIConnect.File.Refresh = 0;
					ActSubState = 4;
					break;

				case 4:
					// Check for file
					for(int i = 0; i < sizeof(MpFileManagerUIConnect.File.List.Items)/sizeof(MpFileManagerUIConnect.File.List.Items[0]); i++)
					{
						if(brsstrcmp((UDINT)&MpFileManagerUIConnect.File.List.Items[i].Name, (UDINT)&DirName) == 0)
							NameMatch = 1;
					}
					TestState = 2;
					break;
			}
			break;

		case 2:
			// Check if file was deleted
			TEST_ASSERT(!NameMatch);
			TEST_DONE;
			break;
	}
	TEST_BUSY;
}

_TEST FIFO_20(void)
{
	TEST_DONE;
	switch (TestState)
	{
		// Arrange
		case 0:
			FileCreate_UT.enable = true;
			FileCreate_UT.pDevice = (UDINT)&"mappUserXFiles";
			snprintf2(FileName, sizeof(FileName), "TestFile%d.txt", FileNumber);
			FileCreate_UT.pFile = (UDINT)&FileName;
			FileCreate(&FileCreate_UT);

			TEST_BUSY_CONDITION(FileCreate_UT.status == 65535);
			TEST_ABORT_CONDITION(FileCreate_UT.status != 0);
			TestState = 1;
			break;

		case 1:
			FileClose_UT.enable = true;
			FileClose_UT.ident = FileCreate_UT.ident;
			FileClose(&FileClose_UT);

			TEST_BUSY_CONDITION(FileClose_UT.status == 65535);
			TEST_ABORT_CONDITION(FileClose_UT.status != 0);

			FileNumber++;
			TestState = (FileNumber >= 20) ? 10 : 0;
			break;

		// Act
		case 10:
			HmiFile_UT.Parameters.Fifo.Enable = true;
			strcpy(HmiFile_UT.Parameters.Fifo.DeviceName, "mappUserXFiles");
			HmiFile_UT.Parameters.Fifo.FifoType = FILE_FIFO_NUM_OF_FILES;
			HmiFile_UT.Parameters.Fifo.MaxNumberOfFiles = 10;
			HmiFile_UT.Parameters.Fifo.ScanInterval = 0;
			TEST_BUSY_CONDITION(FileIdleOrDisabled());
			TestState = 100;
			break;

		// Assert
		case 100:
			TEST_BUSY_CONDITION(!FileIdleOrDisabled());
			HmiFile_UT.Parameters.Fifo.Enable = false;

			DirInfo_UT.enable = true;
			DirInfo_UT.pDevice = (UDINT)&"mappUserXFiles";
			DirInfo_UT.pPath = (UDINT)&"";
			DirInfo(&DirInfo_UT);
			TEST_BUSY_CONDITION(DirInfo_UT.status == 65535);
			TEST_ABORT_CONDITION(DirInfo_UT.status != 0);
			TEST_ASSERT_EQUAL_INT(HmiFile_UT.Parameters.Fifo.MaxNumberOfFiles, DirInfo_UT.filenum);
			TEST_DONE;
			break;
	}
	TEST_BUSY;
}

_TEST FIFO_60(void)
{
	TEST_DONE;
	switch (TestState)
	{
		// Arrange
		case 0:
			FileCreate_UT.enable = true;
			FileCreate_UT.pDevice = (UDINT)&"mappUserXFiles";
			snprintf2(FileName, sizeof(FileName), "TestFile%d.txt", FileNumber);
			FileCreate_UT.pFile = (UDINT)&FileName;
			FileCreate(&FileCreate_UT);

			TEST_BUSY_CONDITION(FileCreate_UT.status == 65535);
			TEST_ABORT_CONDITION(FileCreate_UT.status != 0);
			TestState = 1;
			break;

		case 1:
			FileClose_UT.enable = true;
			FileClose_UT.ident = FileCreate_UT.ident;
			FileClose(&FileClose_UT);

			TEST_BUSY_CONDITION(FileClose_UT.status == 65535);
			TEST_ABORT_CONDITION(FileClose_UT.status != 0);

			FileNumber++;
			TestState = (FileNumber >= 60) ? 10 : 0;
			break;

		// Act
		case 10:
			HmiFile_UT.Parameters.Fifo.Enable = true;
			strcpy(HmiFile_UT.Parameters.Fifo.DeviceName, "mappUserXFiles");
			HmiFile_UT.Parameters.Fifo.FifoType = FILE_FIFO_NUM_OF_FILES;
			HmiFile_UT.Parameters.Fifo.MaxNumberOfFiles = 15;
			HmiFile_UT.Parameters.Fifo.ScanInterval = 0;
			TEST_BUSY_CONDITION(FileIdleOrDisabled());
			TestState = 100;
			break;

		// Assert
		case 100:
			TEST_BUSY_CONDITION(!FileIdleOrDisabled());
			HmiFile_UT.Parameters.Fifo.Enable = false;

			DirInfo_UT.enable = true;
			DirInfo_UT.pDevice = (UDINT)&"mappUserXFiles";
			DirInfo_UT.pPath = (UDINT)&"";
			DirInfo(&DirInfo_UT);
			TEST_BUSY_CONDITION(DirInfo_UT.status == 65535);
			TEST_ABORT_CONDITION(DirInfo_UT.status != 0);
			TEST_ASSERT_EQUAL_INT(HmiFile_UT.Parameters.Fifo.MaxNumberOfFiles, DirInfo_UT.filenum);
			TEST_DONE;
			break;

	}
	TEST_BUSY;
}

_TEST FIFO_140(void)
{
	TEST_DONE;
	switch (TestState)
	{
		// Arrange
		case 0:
			FileCreate_UT.enable = true;
			FileCreate_UT.pDevice = (UDINT)&"mappUserXFiles";
			snprintf2(FileName, sizeof(FileName), "TestFile%d.txt", FileNumber);
			FileCreate_UT.pFile = (UDINT)&FileName;
			FileCreate(&FileCreate_UT);

			TEST_BUSY_CONDITION(FileCreate_UT.status == 65535);
			TEST_ABORT_CONDITION(FileCreate_UT.status != 0);
			TestState = 1;
			break;

		case 1:
			FileClose_UT.enable = true;
			FileClose_UT.ident = FileCreate_UT.ident;
			FileClose(&FileClose_UT);

			TEST_BUSY_CONDITION(FileClose_UT.status == 65535);
			TEST_ABORT_CONDITION(FileClose_UT.status != 0);

			FileNumber++;
			TestState = (FileNumber >= 140) ? 10 : 0;
			break;

		// Act
		case 10:
			HmiFile_UT.Parameters.Fifo.Enable = true;
			strcpy(HmiFile_UT.Parameters.Fifo.DeviceName, "mappUserXFiles");
			HmiFile_UT.Parameters.Fifo.FifoType = FILE_FIFO_NUM_OF_FILES;
			HmiFile_UT.Parameters.Fifo.MaxNumberOfFiles = 15;
			HmiFile_UT.Parameters.Fifo.ScanInterval = 0;
			TEST_BUSY_CONDITION(FileIdleOrDisabled());
			TestState = 100;
			break;

		// Assert
		case 100:
			TEST_BUSY_CONDITION(!FileIdleOrDisabled());
			HmiFile_UT.Parameters.Fifo.Enable = false;

			DirInfo_UT.enable = true;
			DirInfo_UT.pDevice = (UDINT)&"mappUserXFiles";
			DirInfo_UT.pPath = (UDINT)&"";
			DirInfo(&DirInfo_UT);
			TEST_BUSY_CONDITION(DirInfo_UT.status == 65535);
			TEST_ABORT_CONDITION(DirInfo_UT.status != 0);
			TEST_ASSERT_EQUAL_INT(HmiFile_UT.Parameters.Fifo.MaxNumberOfFiles, DirInfo_UT.filenum);
			TEST_DONE;
			break;

	}
	TEST_BUSY;
}

_TEST FIFO_MaxFiles60(void)
{
	TEST_DONE;
	switch (TestState)
	{
		// Arrange
		case 0:
			FileCreate_UT.enable = true;
			FileCreate_UT.pDevice = (UDINT)&"mappUserXFiles";
			snprintf2(FileName, sizeof(FileName), "TestFile%d.txt", FileNumber);
			FileCreate_UT.pFile = (UDINT)&FileName;
			FileCreate(&FileCreate_UT);

			TEST_BUSY_CONDITION(FileCreate_UT.status == 65535);
			TEST_ABORT_CONDITION(FileCreate_UT.status != 0);
			TestState = 1;
			break;

		case 1:
			FileClose_UT.enable = true;
			FileClose_UT.ident = FileCreate_UT.ident;
			FileClose(&FileClose_UT);

			TEST_BUSY_CONDITION(FileClose_UT.status == 65535);
			TEST_ABORT_CONDITION(FileClose_UT.status != 0);

			FileNumber++;
			TestState = (FileNumber >= 100) ? 10 : 0;
			break;

		// Act
		case 10:
			HmiFile_UT.Parameters.Fifo.Enable = true;
			strcpy(HmiFile_UT.Parameters.Fifo.DeviceName, "mappUserXFiles");
			HmiFile_UT.Parameters.Fifo.FifoType = FILE_FIFO_NUM_OF_FILES;
			HmiFile_UT.Parameters.Fifo.MaxNumberOfFiles = 60;
			HmiFile_UT.Parameters.Fifo.ScanInterval = 0;
			TEST_BUSY_CONDITION(FileIdleOrDisabled());
			TestState = 100;
			break;

		// Assert
		case 100:
			TEST_BUSY_CONDITION(!FileIdleOrDisabled());
			HmiFile_UT.Parameters.Fifo.Enable = false;

			DirInfo_UT.enable = true;
			DirInfo_UT.pDevice = (UDINT)&"mappUserXFiles";
			DirInfo_UT.pPath = (UDINT)&"";
			DirInfo(&DirInfo_UT);
			TEST_BUSY_CONDITION(DirInfo_UT.status == 65535);
			TEST_ABORT_CONDITION(DirInfo_UT.status != 0);
			TEST_ASSERT_EQUAL_INT(HmiFile_UT.Parameters.Fifo.MaxNumberOfFiles, DirInfo_UT.filenum);
			TEST_DONE;
			break;

	}
	TEST_BUSY;
}

_TEST FIFO_MaxFiles120(void)
{
	TEST_DONE;
	switch (TestState)
	{
		// Arrange
		case 0:
			FileCreate_UT.enable = true;
			FileCreate_UT.pDevice = (UDINT)&"mappUserXFiles";
			snprintf2(FileName, sizeof(FileName), "TestFile%d.txt", FileNumber);
			FileCreate_UT.pFile = (UDINT)&FileName;
			FileCreate(&FileCreate_UT);

			TEST_BUSY_CONDITION(FileCreate_UT.status == 65535);
			TEST_ABORT_CONDITION(FileCreate_UT.status != 0);
			TestState = 1;
			break;

		case 1:
			FileClose_UT.enable = true;
			FileClose_UT.ident = FileCreate_UT.ident;
			FileClose(&FileClose_UT);

			TEST_BUSY_CONDITION(FileClose_UT.status == 65535);
			TEST_ABORT_CONDITION(FileClose_UT.status != 0);

			FileNumber++;
			TestState = (FileNumber >= 200) ? 10 : 0;
			break;

		// Act
		case 10:
			HmiFile_UT.Parameters.Fifo.Enable = true;
			strcpy(HmiFile_UT.Parameters.Fifo.DeviceName, "mappUserXFiles");
			HmiFile_UT.Parameters.Fifo.FifoType = FILE_FIFO_NUM_OF_FILES;
			HmiFile_UT.Parameters.Fifo.MaxNumberOfFiles = 120;
			HmiFile_UT.Parameters.Fifo.ScanInterval = 0;
			TEST_BUSY_CONDITION(FileIdleOrDisabled());
			TestState = 100;
			break;

		// Assert
		case 100:
			TEST_BUSY_CONDITION(!FileIdleOrDisabled());
			HmiFile_UT.Parameters.Fifo.Enable = false;

			DirInfo_UT.enable = true;
			DirInfo_UT.pDevice = (UDINT)&"mappUserXFiles";
			DirInfo_UT.pPath = (UDINT)&"";
			DirInfo(&DirInfo_UT);
			TEST_BUSY_CONDITION(DirInfo_UT.status == 65535);
			TEST_ABORT_CONDITION(DirInfo_UT.status != 0);
			TEST_ASSERT_EQUAL_INT(HmiFile_UT.Parameters.Fifo.MaxNumberOfFiles, DirInfo_UT.filenum);
			TEST_DONE;
			break;

	}
	TEST_BUSY;
}

_TEST FIFO_MaxFolderSize_30Files(void)
{
	TEST_DONE;
	switch (TestState)
	{
		// Arrange
		case 0:
			FileCreate_UT.enable = true;
			FileCreate_UT.pDevice = (UDINT)&"mappUserXFiles";
			snprintf2(FileName, sizeof(FileName), "TestFile%d.txt", FileNumber);
			FileCreate_UT.pFile = (UDINT)&FileName;
			FileCreate(&FileCreate_UT);

			TEST_BUSY_CONDITION(FileCreate_UT.status == 65535);
			TEST_ABORT_CONDITION(FileCreate_UT.status != 0);
			TestState = 1;
			break;

		case 1:
			FileWrite_UT.enable = true;
			FileWrite_UT.ident = FileCreate_UT.ident;
			FileWrite_UT.offset = 0;
			FileWrite_UT.pSrc = (UDINT)&testData;
			FileWrite_UT.len = sizeof(testData);
			FileWrite(&FileWrite_UT);
			TEST_BUSY_CONDITION(FileWrite_UT.status == 65535);
			TEST_ABORT_CONDITION(FileWrite_UT.status != 0);
			TestState = 2;
			break;

		case 2:
			FileClose_UT.enable = true;
			FileClose_UT.ident = FileCreate_UT.ident;
			FileClose(&FileClose_UT);

			TEST_BUSY_CONDITION(FileClose_UT.status == 65535);
			TEST_ABORT_CONDITION(FileClose_UT.status != 0);

			FileNumber++;
			TestState = (FileNumber >= 30) ? 10 : 0;
			break;

		// Act
		case 10:
			HmiFile_UT.Parameters.Fifo.Enable = true;
			strcpy(HmiFile_UT.Parameters.Fifo.DeviceName, "mappUserXFiles");
			HmiFile_UT.Parameters.Fifo.FifoType = FILE_FIFO_SIZE_OF_FOLDER;
			HmiFile_UT.Parameters.Fifo.MaxFolderSize = 20;
			HmiFile_UT.Parameters.Fifo.ScanInterval = 0;
			TEST_BUSY_CONDITION(FileIdleOrDisabled());
			TestState = 100;
			break;

		// Assert
		case 100:
			TEST_BUSY_CONDITION(!FileIdleOrDisabled());
			HmiFile_UT.Parameters.Fifo.Enable = false;

			DirInfo_UT.enable = true;
			DirInfo_UT.pDevice = (UDINT)&"mappUserXFiles";
			DirInfo_UT.pPath = (UDINT)&"";
			DirInfo(&DirInfo_UT);
			TEST_BUSY_CONDITION(DirInfo_UT.status == 65535);
			TEST_ABORT_CONDITION(DirInfo_UT.status != 0);
			TEST_ASSERT_EQUAL_INT(20, DirInfo_UT.filenum);
			TEST_DONE;
			break;

	}
	TEST_BUSY;
}

_TEST FIFO_MaxFolderSize_60Files(void)
{
	TEST_DONE;
	switch (TestState)
	{
		// Arrange
		case 0:
			FileCreate_UT.enable = true;
			FileCreate_UT.pDevice = (UDINT)&"mappUserXFiles";
			snprintf2(FileName, sizeof(FileName), "TestFile%d.txt", FileNumber);
			FileCreate_UT.pFile = (UDINT)&FileName;
			FileCreate(&FileCreate_UT);

			TEST_BUSY_CONDITION(FileCreate_UT.status == 65535);
			TEST_ABORT_CONDITION(FileCreate_UT.status != 0);
			TestState = 1;
			break;

		case 1:
			FileWrite_UT.enable = true;
			FileWrite_UT.ident = FileCreate_UT.ident;
			FileWrite_UT.offset = 0;
			FileWrite_UT.pSrc = (UDINT)&testData;
			FileWrite_UT.len = sizeof(testData);
			FileWrite(&FileWrite_UT);
			TEST_BUSY_CONDITION(FileWrite_UT.status == 65535);
			TEST_ABORT_CONDITION(FileWrite_UT.status != 0);
			TestState = 2;
			break;

		case 2:
			FileClose_UT.enable = true;
			FileClose_UT.ident = FileCreate_UT.ident;
			FileClose(&FileClose_UT);

			TEST_BUSY_CONDITION(FileClose_UT.status == 65535);
			TEST_ABORT_CONDITION(FileClose_UT.status != 0);

			FileNumber++;
			TestState = (FileNumber >= 60) ? 10 : 0;
			break;

		// Act
		case 10:
			HmiFile_UT.Parameters.Fifo.Enable = true;
			strcpy(HmiFile_UT.Parameters.Fifo.DeviceName, "mappUserXFiles");
			HmiFile_UT.Parameters.Fifo.FifoType = FILE_FIFO_SIZE_OF_FOLDER;
			HmiFile_UT.Parameters.Fifo.MaxFolderSize = 40;
			HmiFile_UT.Parameters.Fifo.ScanInterval = 0;
			TEST_BUSY_CONDITION(FileIdleOrDisabled());
			TestState = 100;
			break;

		// Assert
		case 100:
			TEST_BUSY_CONDITION(!FileIdleOrDisabled());
			HmiFile_UT.Parameters.Fifo.Enable = false;

			DirInfo_UT.enable = true;
			DirInfo_UT.pDevice = (UDINT)&"mappUserXFiles";
			DirInfo_UT.pPath = (UDINT)&"";
			DirInfo(&DirInfo_UT);
			TEST_BUSY_CONDITION(DirInfo_UT.status == 65535);
			TEST_ABORT_CONDITION(DirInfo_UT.status != 0);
			TEST_ASSERT_EQUAL_INT(40, DirInfo_UT.filenum);
			TEST_DONE;
			break;

	}
	TEST_BUSY;
}

_TEST FIFO_MaxFolderSize_Keep60Files(void)
{
	TEST_DONE;
	switch (TestState)
	{
		// Arrange
		case 0:
			FileCreate_UT.enable = true;
			FileCreate_UT.pDevice = (UDINT)&"mappUserXFiles";
			snprintf2(FileName, sizeof(FileName), "TestFile%d.txt", FileNumber);
			FileCreate_UT.pFile = (UDINT)&FileName;
			FileCreate(&FileCreate_UT);

			TEST_BUSY_CONDITION(FileCreate_UT.status == 65535);
			TEST_ABORT_CONDITION(FileCreate_UT.status != 0);
			TestState = 1;
			break;

		case 1:
			FileWrite_UT.enable = true;
			FileWrite_UT.ident = FileCreate_UT.ident;
			FileWrite_UT.offset = 0;
			FileWrite_UT.pSrc = (UDINT)&testData;
			FileWrite_UT.len = sizeof(testData);
			FileWrite(&FileWrite_UT);
			TEST_BUSY_CONDITION(FileWrite_UT.status == 65535);
			TEST_ABORT_CONDITION(FileWrite_UT.status != 0);
			TestState = 2;
			break;

		case 2:
			FileClose_UT.enable = true;
			FileClose_UT.ident = FileCreate_UT.ident;
			FileClose(&FileClose_UT);

			TEST_BUSY_CONDITION(FileClose_UT.status == 65535);
			TEST_ABORT_CONDITION(FileClose_UT.status != 0);

			FileNumber++;
			TestState = (FileNumber >= 90) ? 10 : 0;
			break;

		// Act
		case 10:
			HmiFile_UT.Parameters.Fifo.Enable = true;
			strcpy(HmiFile_UT.Parameters.Fifo.DeviceName, "mappUserXFiles");
			HmiFile_UT.Parameters.Fifo.FifoType = FILE_FIFO_SIZE_OF_FOLDER;
			HmiFile_UT.Parameters.Fifo.MaxFolderSize = 60;
			HmiFile_UT.Parameters.Fifo.ScanInterval = 0;
			TEST_BUSY_CONDITION(FileIdleOrDisabled());
			TestState = 100;
			break;

		// Assert
		case 100:
			TEST_BUSY_CONDITION(!FileIdleOrDisabled());
			HmiFile_UT.Parameters.Fifo.Enable = false;

			DirInfo_UT.enable = true;
			DirInfo_UT.pDevice = (UDINT)&"mappUserXFiles";
			DirInfo_UT.pPath = (UDINT)&"";
			DirInfo(&DirInfo_UT);
			TEST_BUSY_CONDITION(DirInfo_UT.status == 65535);
			TEST_ABORT_CONDITION(DirInfo_UT.status != 0);
			TEST_ASSERT_EQUAL_INT(60, DirInfo_UT.filenum);
			TEST_DONE;
			break;

	}
	TEST_BUSY;
}

_TEST FIFO_MaxFolderSize_Keep120Files(void)
{
	TEST_DONE;
	switch (TestState)
	{
		// Arrange
		case 0:
			FileCreate_UT.enable = true;
			FileCreate_UT.pDevice = (UDINT)&"mappUserXFiles";
			snprintf2(FileName, sizeof(FileName), "TestFile%d.txt", FileNumber);
			FileCreate_UT.pFile = (UDINT)&FileName;
			FileCreate(&FileCreate_UT);

			TEST_BUSY_CONDITION(FileCreate_UT.status == 65535);
			TEST_ABORT_CONDITION(FileCreate_UT.status != 0);
			TestState = 1;
			break;

		case 1:
			FileWrite_UT.enable = true;
			FileWrite_UT.ident = FileCreate_UT.ident;
			FileWrite_UT.offset = 0;
			FileWrite_UT.pSrc = (UDINT)&testData;
			FileWrite_UT.len = sizeof(testData);
			FileWrite(&FileWrite_UT);
			TEST_BUSY_CONDITION(FileWrite_UT.status == 65535);
			TEST_ABORT_CONDITION(FileWrite_UT.status != 0);
			TestState = 2;
			break;

		case 2:
			FileClose_UT.enable = true;
			FileClose_UT.ident = FileCreate_UT.ident;
			FileClose(&FileClose_UT);

			TEST_BUSY_CONDITION(FileClose_UT.status == 65535);
			TEST_ABORT_CONDITION(FileClose_UT.status != 0);

			FileNumber++;
			TestState = (FileNumber >= 140) ? 10 : 0;
			break;

		// Act
		case 10:
			HmiFile_UT.Parameters.Fifo.Enable = true;
			strcpy(HmiFile_UT.Parameters.Fifo.DeviceName, "mappUserXFiles");
			HmiFile_UT.Parameters.Fifo.FifoType = FILE_FIFO_SIZE_OF_FOLDER;
			HmiFile_UT.Parameters.Fifo.MaxFolderSize = 120;
			HmiFile_UT.Parameters.Fifo.ScanInterval = 0;
			TEST_BUSY_CONDITION(FileIdleOrDisabled());
			TestState = 100;
			break;

		// Assert
		case 100:
			TEST_BUSY_CONDITION(!FileIdleOrDisabled());
			HmiFile_UT.Parameters.Fifo.Enable = false;

			DirInfo_UT.enable = true;
			DirInfo_UT.pDevice = (UDINT)&"mappUserXFiles";
			DirInfo_UT.pPath = (UDINT)&"";
			DirInfo(&DirInfo_UT);
			TEST_BUSY_CONDITION(DirInfo_UT.status == 65535);
			TEST_ABORT_CONDITION(DirInfo_UT.status != 0);
			TEST_ASSERT_EQUAL_INT(120, DirInfo_UT.filenum);
			TEST_DONE;
			break;

	}
	TEST_BUSY;
}
/*
B+R UnitTest: This is generated code.
Do not edit! Do not move!
Description: UnitTest Testprogramm infrastructure (TestSet).
LastUpdated: 2023-04-03 16:22:59Z
By B+R UnitTest Helper Version: 2.0.1.59
*/
UNITTEST_FIXTURES(fixtures)
{
	new_TestFixture("Create_Directory", Create_Directory),
	new_TestFixture("Add_File", Add_File),
	new_TestFixture("Copy_File", Copy_File),
	new_TestFixture("Copy_Directory", Copy_Directory),
	new_TestFixture("Rename_File", Rename_File),
	new_TestFixture("Rename_Directory", Rename_Directory),
	new_TestFixture("Cut_Paste_File", Cut_Paste_File),
	new_TestFixture("Cut_Paste_Directory", Cut_Paste_Directory),
	new_TestFixture("Multiselect", Multiselect),
	new_TestFixture("Search", Search),
	new_TestFixture("Enter_Folder", Enter_Folder),
	new_TestFixture("Go_Up_Level", Go_Up_Level),
	new_TestFixture("Change_Sort", Change_Sort),
	new_TestFixture("Delete_File", Delete_File),
	new_TestFixture("Delete_Directory", Delete_Directory),
	new_TestFixture("FIFO_20", FIFO_20),
	new_TestFixture("FIFO_60", FIFO_60),
	new_TestFixture("FIFO_140", FIFO_140),
	new_TestFixture("FIFO_MaxFiles60", FIFO_MaxFiles60),
	new_TestFixture("FIFO_MaxFiles120", FIFO_MaxFiles120),
	new_TestFixture("FIFO_MaxFolderSize_30Files", FIFO_MaxFolderSize_30Files),
	new_TestFixture("FIFO_MaxFolderSize_60Files", FIFO_MaxFolderSize_60Files),
	new_TestFixture("FIFO_MaxFolderSize_Keep60Files", FIFO_MaxFolderSize_Keep60Files),
	new_TestFixture("FIFO_MaxFolderSize_Keep120Files", FIFO_MaxFolderSize_Keep120Files),
};

UNITTEST_CALLER_COMPLETE_EXPLICIT(Set_FileMgr, "Set_FileMgr", setupTest, teardownTest, fixtures, setupSet, teardownSet, cyclicSetCaller);
```

### Package Logical/UnitTestVC4/Recipe - Package for mapp Recipe Framework

### Program Logical/UnitTestVC4/Recipe/RecipeMgrUnitTest (ANSIC)

- RecipeMgr.typ (reference to Logical/Infrastructure/VC4/Recipe/RecipeMgr/RecipeMgr.typ)

- RecipeMgr.var (reference to Logical/Infrastructure/VC4/Recipe/RecipeMgr/RecipeMgr.var)

- Set_Common.c (reference to Logical/UnitTestVC4/Common/CommonUT/Set_Common.c)
